IF NOT __ISVALIDREF(_stState)
THEN
  _eCheck                           := PROCESS_CHECK_STATE_REFERENCE_INVALID;
  RETURN;
END_IF
//-------------------------------------------------------------------------------------------------
//-------------------------------------------------------------------------------------------------
// plausibility checks
//-------------------------------------------------------------------------------------------------
IF NOT Check()
THEN
  RETURN;
END_IF
//-------------------------------------------------------------------------------------------------
//-------------------------------------------------------------------------------------------------
// Message device identification
//-------------------------------------------------------------------------------------------------
_stMsg.eDevice                      := e_Device.Process + TO_UINT(_nProcessId);
//-------------------------------------------------------------------------------------------------
//-------------------------------------------------------------------------------------------------
// XtsStation states:
//  - fb_ProcessCollector extends fb_StationCollector: 
//    --> cyclic call of States() for getting station masks
//
//  - sets bit for every XtsStation
//-------------------------------------------------------------------------------------------------
//
States();                           // collect XtsStation state information in masks
//-------------------------------------------------------------------------------------------------
//-------------------------------------------------------------------------------------------------
// process states
//-------------------------------------------------------------------------------------------------
CASE _stState.State
OF
  //-----------------------------------------------------------------------------------------------
  E_PROCESS_STATE.PROCESS_DISABLE:  // default wait state
    //-------------------------------------------------------------------------
    CASE _eStateProgress            // check if all my XtsStations are disabled
    OF
      E_PROGRESS.PROGRESS_INIT:
        IF (_wStateDisable = EXPT(2,_nStationCount)-1)                  // all stations in process range must be disabled at this point
        THEN
          _eStateProgress           := E_PROGRESS.PROGRESS_BUSY;

          IF (_MessageLevel = E_MessageType.eMessageVerbose)
          THEN
            _stMsg.eType            := E_MessageType.eMessageVerbose;
            _stMsg.eSubdevice       := e_Subdevice.Process_ProcessCollector_Cycle;
            _stMsg.iErrorNumber     := _nProcessId;
            _stMsg.sText            := concat(TO_STRING(_stState.State), ': ');
            _stMsg.sText            := concat(_stMsg.sText, TO_STRING(_eStateProgress));
            f_MessageSet(_stMsg);
          END_IF
        END_IF
    END_CASE
    //-------------------------------------------------------------------------
    CASE _eStateProgress            // check for process enable signal
    OF
      E_PROGRESS.PROGRESS_BUSY:
      CASE _stControl.Cmd                                               // check process command
      OF
        E_PROCESS_CTRL.PROCESS_ENABLE:
          _eCmd                     := _stControl.Cmd;                  // copy command from interface to local switch
          _wActivateStation         := _stControl.ActivateStation;      // on enabling of process, copy my active stations from interface

          _eStateProgress           := E_PROGRESS.PROGRESS_INIT;        // switch back sub state
          _stState.State            := E_PROCESS_STATE.PROCESS_ENABLE;  // switch to enable

          IF (_MessageLevel = E_MessageType.eMessageVerbose)
          THEN
            _stMsg.eType            := E_MessageType.eMessageVerbose;
            _stMsg.eSubdevice       := e_Subdevice.Process_ProcessCollector_Cycle;
            _stMsg.iErrorNumber     := _nProcessId;
            _stMsg.sText            := concat(TO_STRING(_stState.State), ': ');
            _stMsg.sText            := concat(_stMsg.sText, TO_STRING(_eStateProgress));
            f_MessageSet(_stMsg);
          END_IF
      END_CASE
    END_CASE
END_CASE
//-------------------------------------------------------------------------------------------------
//-------------------------------------------------------------------------------------------------
CASE _stState.State
OF
  //-----------------------------------------------------------------------------------------------
  E_PROCESS_STATE.PROCESS_ENABLE:   // wait here for process command "allow infeed"
    //-------------------------------------------------------------------------
    CASE _eStateProgress
    OF
      E_PROGRESS.PROGRESS_INIT:
        IF (_wStateEnable = _wActivateStation)                          // all active stations must be enabled
        THEN
          _eStateProgress           := E_PROGRESS.PROGRESS_BUSY;

          IF (_MessageLevel = E_MessageType.eMessageVerbose)
          THEN
            _stMsg.eType            := E_MessageType.eMessageVerbose;
            _stMsg.eSubdevice       := e_Subdevice.Process_ProcessCollector_Cycle;
            _stMsg.iErrorNumber     := _nProcessId;
            _stMsg.sText            := concat(TO_STRING(_stState.State), ': ');
            _stMsg.sText            := concat(_stMsg.sText, TO_STRING(_eStateProgress));
            f_MessageSet(_stMsg);
          END_IF
        END_IF
    END_CASE
    //-------------------------------------------------------------------------
    CASE _eStateProgress
    OF
      E_PROGRESS.PROGRESS_BUSY:
      // check command for further instructions
      CASE _stControl.Cmd
      OF
        E_PROCESS_CTRL.PROCESS_DISABLE:                                 // command decided to switch OFF  
          _eCmd                     := _stControl.Cmd;                  // copy command from interface
          _eStateProgress           := E_PROGRESS.PROGRESS_INIT;        // switch back sub state
          _stState.State            := E_PROCESS_STATE.PROCESS_DISABLE;

          IF (_MessageLevel = E_MessageType.eMessageVerbose)
          THEN
            _stMsg.eType            := E_MessageType.eMessageVerbose;
            _stMsg.eSubdevice       := e_Subdevice.Process_ProcessCollector_Cycle;
            _stMsg.iErrorNumber     := _nProcessId;
            _stMsg.sText            := concat(TO_STRING(_stState.State), ': ');
            _stMsg.sText            := concat(_stMsg.sText, TO_STRING(_eStateProgress));
            f_MessageSet(_stMsg);
          END_IF


        E_PROCESS_CTRL.PROCESS_STATIONS_INFEED:                          // command decided to allow checking the infeed into process
          _eStateProgress           := E_PROGRESS.PROGRESS_INIT;         // switch back sub state
          _stState.State            := E_PROCESS_STATE.PROCESS_STATIONS_INFEED;

          IF (_MessageLevel = E_MessageType.eMessageVerbose)
          THEN
            _stMsg.eType            := E_MessageType.eMessageVerbose;
            _stMsg.eSubdevice       := e_Subdevice.Process_ProcessCollector_Cycle;
            _stMsg.iErrorNumber     := _nProcessId;
            _stMsg.sText            := concat(TO_STRING(_stState.State), ': ');
            _stMsg.sText            := concat(_stMsg.sText, TO_STRING(_eStateProgress));
            f_MessageSet(_stMsg);
          END_IF
      END_CASE
    END_CASE
END_CASE
//-------------------------------------------------------------------------------------------------
//-------------------------------------------------------------------------------------------------
CASE _stState.State
OF
  //-----------------------------------------------------------------------------------------------
  E_PROCESS_STATE.PROCESS_STATIONS_INFEED:  // wait state for checking infeed command
    //-------------------------------------------------------------------------
    CASE _eStateProgress
    OF
      E_PROGRESS.PROGRESS_INIT:
        IF (_wStateEnter = _wActivateStation)                           // all active XtsStations must have mover waiting
        THEN
          // mover IDs are known by now --> Check _nMoverIdQueue for your plausibility checks
          _eStateProgress           := E_PROGRESS.PROGRESS_BUSY;

          IF (_MessageLevel = E_MessageType.eMessageVerbose)
          THEN
            _stMsg.eType            := E_MessageType.eMessageVerbose;
            _stMsg.eSubdevice       := e_Subdevice.Process_ProcessCollector_Cycle;
            _stMsg.iErrorNumber     := _nProcessId;
            _stMsg.sText            := concat(TO_STRING(_stState.State), ': ');
            _stMsg.sText            := concat(_stMsg.sText, TO_STRING(_eStateProgress));
            f_MessageSet(_stMsg);
          END_IF
        END_IF
    END_CASE
    //-------------------------------------------------------------------------
    CASE _eStateProgress
    OF
      E_PROGRESS.PROGRESS_BUSY:
      CASE _stControl.Cmd                                               // check command from interface
      OF
        E_PROCESS_CTRL.PROCESS_STATIONS_ENTER:
          _eCmd                     := _stControl.Cmd;                  // copy command to start infeed of movers

          _eStateProgress           := E_PROGRESS.PROGRESS_INIT;        // switch back sub state
          _stState.State            := E_PROCESS_STATE.PROCESS_START;

          IF (_MessageLevel = E_MessageType.eMessageVerbose)
          THEN
            _stMsg.eType            := E_MessageType.eMessageVerbose;
            _stMsg.eSubdevice       := e_Subdevice.Process_ProcessCollector_Cycle;
            _stMsg.iErrorNumber     := _nProcessId;
            _stMsg.sText            := concat(TO_STRING(_stState.State), ': ');
            _stMsg.sText            := concat(_stMsg.sText, TO_STRING(_eStateProgress));
            f_MessageSet(_stMsg);
          END_IF


        E_PROCESS_CTRL.PROCESS_STATIONS_SEND:
          _eCmd                     := _stControl.Cmd;                  // start skipping of process

          _eStateProgress           := E_PROGRESS.PROGRESS_INIT;        // switch back sub state
          _stState.State            := E_PROCESS_STATE.PROCESS_STATIONS_OUTFEED;

          IF (_MessageLevel = E_MessageType.eMessageVerbose)
          THEN
            _stMsg.eType            := E_MessageType.eMessageVerbose;
            _stMsg.eSubdevice       := e_Subdevice.Process_ProcessCollector_Cycle;
            _stMsg.iErrorNumber     := _nProcessId;
            _stMsg.sText            := concat(TO_STRING(_stState.State), ': ');
            _stMsg.sText            := concat(_stMsg.sText, TO_STRING(_eStateProgress));
            f_MessageSet(_stMsg);
          END_IF
      END_CASE
    END_CASE
END_CASE
//-------------------------------------------------------------------------------------------------
//-------------------------------------------------------------------------------------------------
CASE _stState.State
OF
  //-----------------------------------------------------------------------------------------------
  E_PROCESS_STATE.PROCESS_STATIONS_NEST:  // wait state before movers are positioned to next nest
    //-------------------------------------------------------------------------
    CASE _eStateProgress
    OF
      E_PROGRESS.PROGRESS_INIT:
        IF (_wStateNest = _wActivateStation)
        THEN
          _eStateProgress           := E_PROGRESS.PROGRESS_BUSY;

          IF (_MessageLevel = E_MessageType.eMessageVerbose)
          THEN
            _stMsg.eType            := E_MessageType.eMessageVerbose;
            _stMsg.eSubdevice       := e_Subdevice.Process_ProcessCollector_Cycle;
            _stMsg.iErrorNumber     := _nProcessId;
            _stMsg.sText            := concat(TO_STRING(_stState.State), ': ');
            _stMsg.sText            := concat(_stMsg.sText, TO_STRING(_eStateProgress));
            f_MessageSet(_stMsg);
          END_IF
        END_IF
    END_CASE
    //-------------------------------------------------------------------------
    CASE _eStateProgress
    OF
      E_PROGRESS.PROGRESS_BUSY:
      CASE _stControl.Cmd
      OF
        E_PROCESS_CTRL.PROCESS_STATIONS_ENTER:
          _eCmd                     := _stControl.Cmd;                  // copy command to start movement to next nest

          _eStateProgress           := E_PROGRESS.PROGRESS_INIT;        // switch back sub state
          _stState.State            := E_PROCESS_STATE.PROCESS_START;

          IF (_MessageLevel = E_MessageType.eMessageVerbose)
          THEN
            _stMsg.eType            := E_MessageType.eMessageVerbose;
            _stMsg.eSubdevice       := e_Subdevice.Process_ProcessCollector_Cycle;
            _stMsg.iErrorNumber     := _nProcessId;
            _stMsg.sText            := concat(TO_STRING(_stState.State), ': ');
            _stMsg.sText            := concat(_stMsg.sText, TO_STRING(_eStateProgress));
            f_MessageSet(_stMsg);
          END_IF
      END_CASE
    END_CASE
END_CASE
//-------------------------------------------------------------------------------------------------
//-------------------------------------------------------------------------------------------------
CASE _stState.State
OF
  //-----------------------------------------------------------------------------------------------
  E_PROCESS_STATE.PROCESS_START:    // wait state for movers to arrive
    //-------------------------------------------------------------------------
    CASE _eStateProgress
    OF
      E_PROGRESS.PROGRESS_INIT:
        IF (_wStateStart = _wActivateStation)                           // all active XtsStations have mover in standstill after infeed, process handshake may now start
        THEN
          // movers have arrived and are in standstill
          _eStateProgress           := E_PROGRESS.PROGRESS_BUSY;

          IF (_MessageLevel = E_MessageType.eMessageVerbose)
          THEN
            _stMsg.eType            := E_MessageType.eMessageVerbose;
            _stMsg.eSubdevice       := e_Subdevice.Process_ProcessCollector_Cycle;
            _stMsg.iErrorNumber     := _nProcessId;
            _stMsg.sText            := concat(TO_STRING(_stState.State), ': ');
            _stMsg.sText            := concat(_stMsg.sText, TO_STRING(_eStateProgress));
            f_MessageSet(_stMsg);
          END_IF
        END_IF
    END_CASE
    //-------------------------------------------------------------------------
    CASE _eStateProgress
    OF
      E_PROGRESS.PROGRESS_BUSY:
      CASE _stControl.Cmd
      OF
        E_PROCESS_CTRL.PROCESS_START:
          _eCmd                     := _stControl.Cmd;                  // first handshake for starting process

          _eStateProgress           := E_PROGRESS.PROGRESS_INIT;        // switch back sub state
          _stState.State            := E_PROCESS_STATE.PROCESS_DONE;

          IF (_MessageLevel = E_MessageType.eMessageVerbose)
          THEN
            _stMsg.eType            := E_MessageType.eMessageVerbose;
            _stMsg.eSubdevice       := e_Subdevice.Process_ProcessCollector_Cycle;
            _stMsg.iErrorNumber     := _nProcessId;
            _stMsg.sText            := concat(TO_STRING(_stState.State), ': ');
            _stMsg.sText            := concat(_stMsg.sText, TO_STRING(_eStateProgress));
            f_MessageSet(_stMsg);
          END_IF
      END_CASE
    END_CASE
END_CASE
//-------------------------------------------------------------------------------------------------
//-------------------------------------------------------------------------------------------------
CASE _stState.State
OF
  E_PROCESS_STATE.PROCESS_DONE:     // wait state for process done
    //-------------------------------------------------------------------------
    CASE _eStateProgress
    OF
      E_PROGRESS.PROGRESS_INIT:
        IF (_wStateDone = _wActivateStation)
        THEN
          // first handshake done
          _eStateProgress           := E_PROGRESS.PROGRESS_BUSY;

          IF (_MessageLevel = E_MessageType.eMessageVerbose)
          THEN
            _stMsg.eType            := E_MessageType.eMessageVerbose;
            _stMsg.eSubdevice       := e_Subdevice.Process_ProcessCollector_Cycle;
            _stMsg.iErrorNumber     := _nProcessId;
            _stMsg.sText            := concat(TO_STRING(_stState.State), ': ');
            _stMsg.sText            := concat(_stMsg.sText, TO_STRING(_eStateProgress));
            f_MessageSet(_stMsg);
          END_IF
        END_IF
    END_CASE
    //-------------------------------------------------------------------------
    CASE _eStateProgress
    OF
      E_PROGRESS.PROGRESS_BUSY:
      CASE _stControl.Cmd
      OF
        E_PROCESS_CTRL.PROCESS_DONE:
          _eCmd                     := _stControl.Cmd;                  // second handshake for finishing process

          _eStateProgress           := E_PROGRESS.PROGRESS_CHECK;       // check mover after process done
      END_CASE
    //-------------------------------------------------------------------------
      E_PROGRESS.PROGRESS_CHECK:
        IF (_wStateNest > 0)        // mover has to be worked again
        THEN
          _eStateProgress           := E_PROGRESS.PROGRESS_INIT;        // switch back sub state
          _stState.State            := E_PROCESS_STATE.PROCESS_STATIONS_NEST;

          IF (_MessageLevel = E_MessageType.eMessageVerbose)
          THEN
            _stMsg.eType            := E_MessageType.eMessageVerbose;
            _stMsg.eSubdevice       := e_Subdevice.Process_ProcessCollector_Cycle;
            _stMsg.iErrorNumber     := _nProcessId;
            _stMsg.sText            := concat(TO_STRING(_stState.State), ': ');
            _stMsg.sText            := concat(_stMsg.sText, TO_STRING(_eStateProgress));
            f_MessageSet(_stMsg);
          END_IF

        ELSIF (_wStateOut > 0)      // mover has to leave
        THEN
          _eStateProgress           := E_PROGRESS.PROGRESS_INIT;        // switch back sub state
          _stState.State            := E_PROCESS_STATE.PROCESS_STATIONS_OUTFEED;

          IF (_MessageLevel = E_MessageType.eMessageVerbose)
          THEN
            _stMsg.eType            := E_MessageType.eMessageVerbose;
            _stMsg.eSubdevice       := e_Subdevice.Process_ProcessCollector_Cycle;
            _stMsg.iErrorNumber     := _nProcessId;
            _stMsg.sText            := concat(TO_STRING(_stState.State), ': ');
            _stMsg.sText            := concat(_stMsg.sText, TO_STRING(_eStateProgress));
            f_MessageSet(_stMsg);
          END_IF
        END_IF
    END_CASE
END_CASE
//-------------------------------------------------------------------------------------------------
//-------------------------------------------------------------------------------------------------
CASE _stState.State
OF
  E_PROCESS_STATE.PROCESS_STATIONS_OUTFEED:   // wait state before movers are sent out
    //-------------------------------------------------------------------------
    CASE _eStateProgress
    OF
      E_PROGRESS.PROGRESS_INIT:
        IF (_wStateOut = _wActivateStation)
        THEN
          // all active stations want to send out mover
          // now is the time for you to have decided the TargetStation(s) and TargetMask(s)
          _eStateProgress           := E_PROGRESS.PROGRESS_BUSY;

          IF (_MessageLevel = E_MessageType.eMessageVerbose)
          THEN
            _stMsg.eType            := E_MessageType.eMessageVerbose;
            _stMsg.eSubdevice       := e_Subdevice.Process_ProcessCollector_Cycle;
            _stMsg.iErrorNumber     := _nProcessId;
            _stMsg.sText            := concat(TO_STRING(_stState.State), ': ');
            _stMsg.sText            := concat(_stMsg.sText, TO_STRING(_eStateProgress));
            f_MessageSet(_stMsg);
          END_IF
        END_IF
    END_CASE
    //-------------------------------------------------------------------------
    CASE _eStateProgress
    OF
      E_PROGRESS.PROGRESS_BUSY:     // now is the time to get/write target data
      CASE _stControl.Cmd
      OF
        E_PROCESS_CTRL.PROCESS_STATIONS_OUTFEED:  // before you start the outfeed of station, get/write target data on the outside. Use properties: TargetIndex; TargetMask
          _eCmd                     := _stControl.Cmd;
          _eStateProgress           := E_PROGRESS.PROGRESS_CHECK;       // check movers gone

          IF (_MessageLevel = E_MessageType.eMessageVerbose)
          THEN
            _stMsg.eType            := E_MessageType.eMessageVerbose;
            _stMsg.eSubdevice       := e_Subdevice.Process_ProcessCollector_Cycle;
            _stMsg.iErrorNumber     := _nProcessId;
            _stMsg.sText            := concat(TO_STRING(_stState.State), ': ');
            _stMsg.sText            := concat(_stMsg.sText, TO_STRING(_eStateProgress));
            f_MessageSet(_stMsg);
          END_IF
      END_CASE
    END_CASE
    //-------------------------------------------------------------------------
    CASE _eStateProgress
    OF
      E_PROGRESS.PROGRESS_CHECK:
        IF (_wStateOut = 0)         // all stations are empty, go back to start new infeed of movers
        THEN
          _eStateProgress           := E_PROGRESS.PROGRESS_INIT;        // switch back sub state
          _stState.State            := E_PROCESS_STATE.PROCESS_DISABLE; // switch back to disabled state

          IF (_MessageLevel = E_MessageType.eMessageVerbose)
          THEN
            _stMsg.eType            := E_MessageType.eMessageVerbose;
            _stMsg.eSubdevice       := e_Subdevice.Process_ProcessCollector_Cycle;
            _stMsg.iErrorNumber     := _nProcessId;
            _stMsg.sText            := concat(TO_STRING(_stState.State), ': ');
            _stMsg.sText            := concat(_stMsg.sText, TO_STRING(_eStateProgress));
            f_MessageSet(_stMsg);
          END_IF
        END_IF
    END_CASE
END_CASE
//-------------------------------------------------------------------------------------------------
// _eStateProgress information to process result
//-------------------------------------------------------------------------------------------------
_stState.Result                     := _eStateProgress;
//-------------------------------------------------------------------------------------------------
//-------------------------------------------------------------------------------------------------
// _eCheck information for plausibility checks
//-------------------------------------------------------------------------------------------------
_stState.Check                      := _eCheck;
//-------------------------------------------------------------------------------------------------
//-------------------------------------------------------------------------------------------------
// _eCmd - command switch
//-------------------------------------------------------------------------------------------------
Controls(_eCmd);                    // cyclic call for setting commands on XtsStations in process range
//-------------------------------------------------------------------------------------------------
//-------------------------------------------------------------------------------------------------
END_METHOD

METHOD PUBLIC Init : E_PROGRESS // clears all XtsSubstations, then disables all
VAR_INPUT
  Execute     : BOOL;
END_VAR
VAR_INST
  _nIndexStation        : UINT;
  _nErrorId             : UDINT;
  _eState               : E_PROGRESS;
END_VAR
//-----------------------------------------------------------------------------
IF NOT Execute 
THEN 
	_eState                       := E_PROGRESS.PROGRESS_INIT; 
END_IF 
//-----------------------------------------------------------------------------
IF NOT Check() 
THEN 
	Init                          := E_PROGRESS.PROGRESS_ERROR; 
	RETURN; 
END_IF
//-----------------------------------------------------------------------------
//-----------------------------------------------------------------------------
CASE _eState
OF
  E_PROGRESS.PROGRESS_INIT:
    IF Execute
    THEN
      _nIndexStation            := _nStationLast;
      _nErrorId                 := 0;
      _eState                   := E_PROGRESS.PROGRESS_BUSY;
      memset(ADR(_wTargetMask), 1, SIZEOF(_wTargetMask));

      _eCmd                     := E_PROCESS_CTRL.PROCESS_INIT;
      _stState.State            := E_PROCESS_STATE.PROCESS_INVALID;
      _eStateProgress           := E_PROGRESS.PROGRESS_INVALID;


      _stMsg.eType              := _MessageLevel;

      IF (_MessageLevel = E_MessageType.eMessageVerbose)
      THEN
        _stMsg.eSubdevice       := e_Subdevice.Process_ProcessCollector_Init;
        _stMsg.iErrorNumber     := _nIndexStation;
        _stMsg.sText            := concat('.Init: ', TO_STRING(_eState));
        f_MessageSet(_stMsg);
      END_IF
    END_IF
END_CASE
//-----------------------------------------------------------------------------
//-----------------------------------------------------------------------------
CASE _eState
OF
  E_PROGRESS.PROGRESS_BUSY:
    _StationCtrl[_nIndexStation].eCmd     := E_STATION_CTRL.STATION_INIT;
    _eState                     := E_PROGRESS.PROGRESS_PREPARE;

    IF (_MessageLevel = E_MessageType.eMessageVerbose)
    THEN
      _stMsg.eSubdevice         := e_Subdevice.Process_ProcessCollector_Init;
      _stMsg.iErrorNumber       := _nIndexStation;
      _stMsg.sText              := concat(TO_STRING(_StationCtrl[_nIndexStation].eCmd), ': ');
      _stMsg.sText              := concat(_stMsg.sText, TO_STRING(_eState));
      f_MessageSet(_stMsg);
    END_IF

  E_PROGRESS.PROGRESS_PREPARE:
    IF (_nIndexStation < _nStationFirst+1)
    THEN
      _eCmdOld                  :=
      _eCmd                     := E_PROCESS_CTRL.PROCESS_DISABLE;
      _nIndexStation            := _nStationFirst;
      _eState                   := E_PROGRESS.PROGRESS_STARTUP;
    ELSE
      IF (_StationState[_nIndexStation].eState = E_STATION_STATE.STATION_INIT)
      THEN
        _nIndexStation          := _nIndexStation - 1;
        _eState                 := E_PROGRESS.PROGRESS_BUSY;
      ELSE
        _eState                 := E_PROGRESS.PROGRESS_BUSY;
      END_IF
    END_IF

  E_PROGRESS.PROGRESS_STARTUP:
    _StationCtrl[_nIndexStation].eCmd     := E_STATION_CTRL.STATION_DISABLE;
    _eState                     := E_PROGRESS.PROGRESS_CHECK;

    IF (_MessageLevel = E_MessageType.eMessageVerbose)
    THEN
      _stMsg.eSubdevice         := e_Subdevice.Process_ProcessCollector_Init;
      _stMsg.iErrorNumber       := _nIndexStation;
      _stMsg.sText              := concat(TO_STRING(_StationCtrl[_nIndexStation].eCmd), ': ');
      _stMsg.sText              := concat(_stMsg.sText, TO_STRING(_eState));
      f_MessageSet(_stMsg);
    END_IF

  E_PROGRESS.PROGRESS_CHECK:
    IF NOT (_nIndexStation > _nStationLast-1)
    THEN
      IF (_StationState[_nIndexStation].eState = E_STATION_STATE.STATION_DISABLE)
      THEN
        _nIndexStation          := _nIndexStation + 1;
        _eState                 := E_PROGRESS.PROGRESS_STARTUP;
      END_IF
    ELSE
      // give back result
      _eState                   := E_PROGRESS.PROGRESS_DONE;

      // where were I?
      IF (_MessageLevel = E_MessageType.eMessageVerbose)
      THEN
        _stMsg.eSubdevice       := e_Subdevice.Process_ProcessCollector_Init;
        _stMsg.iErrorNumber     := _nProcessId;
        _stMsg.sText            := concat('.Clear: ', TO_STRING(_stState.State));
        f_MessageSet(_stMsg);
      END_IF

      // clear Cycle() state machine
      _stState.State            := E_PROCESS_STATE.PROCESS_DISABLE;
      _eStateProgress           := E_PROGRESS.PROGRESS_INIT;

      IF (_MessageLevel = E_MessageType.eMessageVerbose)
      THEN
        // init done
        _stMsg.eSubdevice       := e_Subdevice.Process_ProcessCollector_Init;
        _stMsg.iErrorNumber     := _nProcessId;
        _stMsg.sText            := concat('.Init: ', TO_STRING(_eState));
        f_MessageSet(_stMsg);
      END_IF
    END_IF
END_CASE
//-----------------------------------------------------------------------------
//-----------------------------------------------------------------------------

Init := _eState;
END_METHOD

PROPERTY MessageLevel : e_MessageType
GET
MessageLevel := _MessageLevel;
END_GET
SET
VAR
  _ix : uint;
END_VAR
_MessageLevel := MessageLevel;

IF NOT (_eCheck = E_PROCESS_CHECK.PROCESS_CHECK_DONE)
THEN
  RETURN;
ELSE
  FOR _ix := _nStationFirst TO _nStationLast
  DO
    GVL_MSG.MessageLevelStations[_ix]   := _MessageLevel;
  END_FOR
END_IF
END_SET
END_PROPERTY

PROPERTY MoverCountTotal : udint
GET
MoverCountTotal := _nMoverCountTotal;
END_GET
END_PROPERTY

PROPERTY MoverPerMinute : udint
GET
MoverPerMinute := _AllStationMoverPerMinute;
END_GET
END_PROPERTY

PROPERTY ProcessCtrl : reference to st_process_ctrl
GET
ProcessCtrl REF= _stControl;
END_GET
SET
_stControl ref= ProcessCtrl;
END_SET
END_PROPERTY

PROPERTY ProcessId : E_INSTANCE
GET
Processid := _nProcessId;
END_GET
SET
_nProcessId := ProcessId;
END_SET
END_PROPERTY

PROPERTY ProcessState : reference to st_process_state
GET
ProcessState REF= _stState;
END_GET
SET
_stState ref= ProcessState;
END_SET
END_PROPERTY

PROPERTY TargetIndex : ARRAY[1..SIZEOF(T_PROCESS)*8] OF USINT
GET
TargetIndex := _nTargetIndex;
END_GET
SET
_nTargetIndex := TargetIndex;
END_SET
END_PROPERTY

PROPERTY TargetMask : ARRAY[1..SIZEOF(T_PROCESS)*8] OF BYTE
GET
TargetMask := _wTargetMask;
END_GET
SET
_wTargetMask := TargetMask;
END_SET
END_PROPERTY

METHOD Template : E_PROGRESS
VAR_INPUT
  Execute     : BOOL;
END_VAR
VAR_INST
  _nErrorId   : UDINT;
  _eState     : E_PROGRESS;
END_VAR
//-----------------------------------------------------------------------------
IF NOT Execute 
THEN 
	_eState                       := E_PROGRESS.PROGRESS_INIT; 
END_IF 
//-----------------------------------------------------------------------------
IF NOT Check() 
THEN 
	Template_1                    := E_PROGRESS.PROGRESS_ERROR; 
	RETURN; 
END_IF
//-----------------------------------------------------------------------------
//-----------------------------------------------------------------------------
CASE _eState
OF
  E_PROGRESS.PROGRESS_INIT:
    IF Execute
    THEN
      _nErrorId                 := 0;

      _eState                   := E_PROGRESS.PROGRESS_BUSY;
    END_IF
END_CASE
//-----------------------------------------------------------------------------
//-----------------------------------------------------------------------------
CASE _eState
OF
  E_PROGRESS.PROGRESS_BUSY:
    _eState                     := E_PROGRESS.PROGRESS_PREPARE;
END_CASE
//-----------------------------------------------------------------------------
//-----------------------------------------------------------------------------
CASE _eState
OF
  E_PROGRESS.PROGRESS_PREPARE:

    IF (.Error)
    THEN
      _eState                   := E_PROGRESS.PROGRESS_ERROR;
      _nErrorId                 := 


    ELSIF (.Done)
    THEN
      _eState                   := E_PROGRESS.;

    END_IF
END_CASE
//-----------------------------------------------------------------------------
//-----------------------------------------------------------------------------

Template_1                      := _eState;
END_METHOD

END_FUNCTION_BLOCK

// ---- XTS/XtsStation/fb_Station.TcPOU
//---------------------------------------------------------------------------------------------------------------
//
//  HAUD 2023.03.07
//
//  - XTS_TRANSPORT_LAYER
//
//  fb_Station
//  - handshake with extern control for mover transport through station
//
//---------------------------------------------------------------------------------------------------------------
// This SOFTWARE is provided as an Exemple by THE PROVIDER "as is" and "with all faults." THE PROVIDER makes no 
// representations or warranties of any kind concerning the safety, suitability, lack of viruses, inaccuracies, 
// typographical errors, or other harmful components of this SOFTWARE. There are inherent dangers in the use of 
// any software, and you are solely responsible for determining whether this SOFTWARE is compatible with your 
// equipment and other software installed on your equipment. You are also solely responsible for the protection 
// of your equipment and backup of your data, and THE PROVIDER will not be liable for any damages you may suffer 
// in connection with using, modifying, or distributing this SOFTWARE.
//---------------------------------------------------------------------------------------------------------------
FUNCTION_BLOCK fb_Station IMPLEMENTS I_XtsTransport_Station
VAR
  _nStationId                 : UINT;         // why is Gamora?

  _sState                     : STRING(255);  // additional output for Check()

  _eInitList                  : E_PROGRESS;   // linked list initialization progress

  _eFatalError                : E_STATION_STATE;

  // pointer to all stations
  _stCtrl                     : REFERENCE TO ARRAY[1..MAX_STATION]  OF ST_STATION_CTRL;
  _stState                    : REFERENCE TO ARRAY[1..MAX_STATION]  OF ST_STATION_STATE;

  // local copy of command
  _eCmd,
  _eCmdOld                    : E_STATION_CTRL;

  _ItfStation                 : REFERENCE TO ARRAY[1..MAX_STATION]  OF I_Station_LinkedList;  // access to all stations lists
  _ItfMover                   : REFERENCE TO ARRAY[1..MAX_MOVER]    OF I_XtsTransport_Mover;  // access to mover methods

  // station related data
  _rMoverOffset               : REFERENCE TO ARRAY[1..MAX_STATION]  OF T_NEST_OFFSET;         // static offsets for station
  _stParameter                : REFERENCE TO ARRAY[1..MAX_STATION]  OF ST_STATION_PARAMETER;  // station parameter (where, how fast, how many stops)

  // mover axis ref for info
  _Mover                      : REFERENCE TO ARRAY[1..MAX_MOVER]    OF AXIS_REF;              // read from AXIS_REF

  // linked list result struct
  _stListEnter,
  _stListTarget,
  _stListDelete               : ST_STATION_LIST_RESULT;   // struct with result and ticket data

  _stMoverDataSend,
  _stMoverData                : ST_STATION_MOVER_DATA;    // mover ticket data

  _stInfeed,
  _stOutfeed                  : ST_MOVE_DATA;             // position and dynamic constraints of movement

  // work vars
  _Result                     : E_PROGRESS;
  _eStateProgress             : E_PROGRESS;

  _nNest,
  _nMoverDetected,
  _ix                         : UINT;

  _rModActPosFetch            : LREAL;
  _stMsg                      : ST_Message;
  _eMessageLevel              : E_MessageType;
  _bMatchMessageLevel         : BOOL := TRUE;   // TRUE --> Mover in Station commands have equal message level as station
END_VAR

METHOD PRIVATE Check : BOOL
VAR_INPUT
END_VAR
IF NOT (_nStationId > 0) OR
       (_nStationId > MAX_STATION)
THEN
  _sState                     := 'invalid nStationId';
  RETURN;
END_IF

IF NOT __ISVALIDREF(_stCtrl)
THEN
  _sState                     := '_stCtrl: missing pointer';
  RETURN;
END_IF

IF NOT __ISVALIDREF(_stState)
THEN
  _sState                     := '_stState: missing pointer';
  RETURN;
END_IF

IF NOT __ISVALIDREF(_ItfStation)
THEN
  _sState                     := '_ItfStation: missing interface';
  RETURN;
END_IF

IF NOT __ISVALIDREF(_ItfMover)
THEN
  _sState                     := '_ItfMover: missing interface';
  RETURN;
END_IF

IF NOT __ISVALIDREF(_rMoverOffset)
THEN
  _sState                     := '_rMoverOffset: missing pointer';
  RETURN;
END_IF

IF NOT __ISVALIDREF(_stParameter)
THEN
  _sState                     := '_stParameter: missing pointer';
  RETURN;
END_IF

IF NOT __ISVALIDREF(_Mover)
THEN
  _sState                     := '_Mover: missing pointer';
  RETURN;
END_IF


_sState                       := 'CHECK_DONE';
Check                         := TRUE;
END_METHOD

PROPERTY Ctrl : reference to ARRAY[1..MAX_STATION] OF ST_STATION_CTRL
SET
_stCtrl ref= Ctrl;
END_SET
END_PROPERTY

METHOD Cycle
//-----------------------------------------------------------------------------
//-----------------------------------------------------------------------------
// check pointer and interface
//-----------------------------------------------------------------------------
IF NOT Check() THEN RETURN; END_IF
//-----------------------------------------------------------------------------
//-----------------------------------------------------------------------------
// set message device ID
//-----------------------------------------------------------------------------
_stMsg.eDevice                        := e_Device.XtsStation + _nStationId;
//-----------------------------------------------------------------------------
//-----------------------------------------------------------------------------
// log command change
//-----------------------------------------------------------------------------
_eCmd                                 := _stCtrl[_nStationId].eCmd;
IF (_eCmd <> _eCmdOld)
THEN
  _eCmdOld                            := _eCmd;

  _stMsg.eType                        := E_MessageType.eMessageInfo;
  _stMsg.eSubdevice                   := StationControl;
  _stMsg.iErrorNumber                 := 0;
  _stMsg.sText                        := TO_STRING(_eCmd);

  IF (_eMessageLevel > E_MessageType.eMessageWarning)
  THEN
    f_MessageSet(_stMsg);
  END_IF
END_IF
//-----------------------------------------------------------------------------
//-----------------------------------------------------------------------------
// clear station on demand
//-----------------------------------------------------------------------------
CASE _stCtrl[_nStationId].eCmd
OF
  E_STATION_CTRL.STATION_INIT:        // commanded init from cyclic interface
    _eInitList                        := Init();
    _stState[_nStationId].rMoverModPos:= 0.0;
    _stState[_nStationId].nQueue      := TO_USINT(_ItfStation[_nStationId].Count);
    RETURN;
END_CASE
//-----------------------------------------------------------------------------
//-----------------------------------------------------------------------------
// station startup and init states
//-----------------------------------------------------------------------------
CASE _stState[_nStationId].eState
OF
  E_STATION_STATE.STATION_NO_INIT:    // startup state in first PLC cycle, init linked list required
    _eInitList                        := Init();

  E_STATION_STATE.STATION_INIT:       // switch state as reserve for anything you might add here
    _stState[_nStationId].eState      := E_STATION_STATE.STATION_DISABLE;
END_CASE
//-----------------------------------------------------------------------------
//-----------------------------------------------------------------------------
//  station disabled after init 
//  wait for command to enable
//  return state after a mover has left station
//  fall back state before entry was allowed and you decided to disable
//-----------------------------------------------------------------------------
CASE _stState[_nStationId].eState
OF
  E_STATION_STATE.STATION_DISABLE:
    IF (_stCtrl[_nStationId].eCmd = E_STATION_CTRL.STATION_ENABLE)
    THEN
      _stState[_nStationId].eState    := E_STATION_STATE.STATION_ENABLE;
    END_IF


  E_STATION_STATE.STATION_ENABLE:     // enable state is detectable on the interface for one cycle only
                                      // double check commanded enable and clear work vars
    IF (_stCtrl[_nStationId].eCmd = E_STATION_CTRL.STATION_ENABLE)
    THEN
      memset(ADR(_stListEnter),    0, SIZEOF(_stListEnter));

      _eStateProgress                 := E_PROGRESS.PROGRESS_INIT;  // substate for procedures within one state
      _stState[_nStationId].eState    := E_STATION_STATE.STATION_DETECT_MOVER;  // switch to mover detection

      IF (_eMessageLevel = E_MessageType.eMessageVerbose)
      THEN
        _stMsg.eType                  := _eMessageLevel;
        LogState(_stMsg.eType);
      END_IF
    END_IF
END_CASE
//-----------------------------------------------------------------------------
//-----------------------------------------------------------------------------
//  detection state
//   - wait until mover data is entered into list
//
//  check for disable command; fall back to disabled state
//  check linked list for new entry; proceed to request infeed of mover
//-----------------------------------------------------------------------------
CASE _stState[_nStationId].eState
OF
  E_STATION_STATE.STATION_DETECT_MOVER:// wait state for mover detection
    CASE _eStateProgress
    OF
      E_PROGRESS.PROGRESS_INIT:
        IF (_stCtrl[_nStationId].eCmd = E_STATION_CTRL.STATION_DISABLE) // check for commanded disable
        THEN
          IF (_eMessageLevel = E_MessageType.eMessageVerbose)
          THEN
            _stMsg.eType              := E_MessageType.eMessageVerbose;
            _stMsg.eSubdevice         := Stationstate;
            _stMsg.iErrorNumber       := _stState[_nStationId].nMoverId;
            _stMsg.sText              := concat(TO_STRING(_stState[_nStationId].eState), ': ');
            _stMsg.sText              := concat(_stMsg.sText, TO_STRING(E_STATION_STATE.STATION_DISABLE));
            f_MessageSet(_stMsg);
          END_IF
          _stState[_nStationId].eState      := E_STATION_STATE.STATION_DISABLE; // go back and wait, no matter the queue

        ELSIF (_ItfStation[_nStationId].Count > 0)
        THEN
          // someone entered something in my list
          _stListEnter                := _ItfStation[_nStationId].GetHead();
          _eStateProgress             := E_PROGRESS.PROGRESS_BUSY;  // go check list result data

          IF (_eMessageLevel > E_MessageType.eMessageWarning)
          THEN
            _stMsg.eType              := E_MessageType.eMessageInfo;
            _stMsg.eSubdevice         := Stationstate;
            _stMsg.iErrorNumber       := _stState[_nStationId].nMoverId;
            _stMsg.sText              := concat(TO_STRING(_stState[_nStationId].eState), ': ');
            _stMsg.sText              := concat(_stMsg.sText, TO_STRING(_eStateProgress));
            f_MessageSet(_stMsg);
          END_IF
        END_IF
    END_CASE
    CASE _eStateProgress
    OF
      E_PROGRESS.PROGRESS_BUSY:
        IF (_stListEnter.wState = 0)  // GetHead() without error
        THEN
          _stMsg.eType                := E_MessageType.eMessageVerbose;
          _stMsg.eSubdevice           := e_Subdevice.StationGetHead;
          _stMsg.iErrorNumber         := _stListEnter.stData.nMoverId;
          _stMsg.sText                := '';
          IF (_eMessageLevel = E_MessageType.eMessageVerbose)
          THEN
            f_MessageSet(_stMsg);
          END_IF

          // list is giving head as result
          _stMoverData                := _stListEnter.stData; // copy ticket from list result
          _eStateProgress             := E_PROGRESS.PROGRESS_PREPARE; // go check plausibility of ticket

          IF (_eMessageLevel = E_MessageType.eMessageVerbose)
          THEN
            _stMsg.eType              := E_MessageType.eMessageVerbose;
            _stMsg.eSubdevice         := Stationstate;
            _stMsg.iErrorNumber       := _stState[_nStationId].nMoverId;
            _stMsg.sText              := concat(TO_STRING(_stState[_nStationId].eState), ': ');
            _stMsg.sText              := concat(_stMsg.sText, TO_STRING(_eStateProgress));
            f_MessageSet(_stMsg);
          END_IF
        ELSE
          // the thing that must not be: GetHead() with error
          _stState[_nStationId].eState      := E_STATION_STATE.STATION_ERROR_LIST_GET_HEAD_FAULT; // fatal error

          _stMsg.eType                      := E_MessageType.eMessageError;
          LogState(_stMsg.eType);
        END_IF
    END_CASE
    CASE _eStateProgress
    OF
      E_PROGRESS.PROGRESS_PREPARE:    // check ticket (list entry)
        // check target assignement
        IF NOT (_stMoverData.nTargetStation = _nStationId)
        THEN
          // for whom the mover calls
          // wrong address, right mover?
          _stState[_nStationId].eState      := E_STATION_STATE.STATION_ERROR_LIST_STATION_ID_WRONG; // ctrl has to fix this, go tell ctrl

          _stMsg.eType                      := E_MessageType.eMessageWarning;
          LogState(_stMsg.eType);
        ELSE
          // it's a me
          _nMoverDetected                   := _stMoverData.nMoverId;

          IF (_nMoverDetected < 1) OR
             (_nMoverDetected > MAX_MOVER)
          THEN
            // out of range the mover must not be
            _stState[_nStationId].eState    := E_STATION_STATE.STATION_ERROR_LIST_MOVER_ID_INVALID; // fatal error

            _stMsg.eType                    := E_MessageType.eMessageError;
            LogState(_stMsg.eType);
          ELSE
            memset(ADR(_stListDelete),   0, SIZEOF(_stListDelete)); // clear work var
            _eStateProgress                 := E_PROGRESS.PROGRESS_INIT; // clear progress for next station state

            // prepare station state for new mover
            _stState[_nStationId].nMoverId  := TO_USINT(_nMoverDetected); // who is waiting to enter
            _stState[_nStationId].nMask     := _stMoverData.nMask;        // how many stops have to be made
            _stState[_nStationId].eState    := E_STATION_STATE.STATION_MOVER_ENTER; // go ask for permission to enter

            IF (_eMessageLevel > E_MessageType.eMessageWarning)
            THEN
              _stMsg.eType            := E_MessageType.eMessageInfo;
              _stMsg.eSubdevice       := Stationstate;
              _stMsg.iErrorNumber     := _stState[_nStationId].nMoverId;
              _stMsg.sText            := concat(TO_STRING(_stState[_nStationId].eState), ': ');
              _stMsg.sText            := concat(_stMsg.sText, TO_STRING(_eStateProgress));
              f_MessageSet(_stMsg);
            END_IF
          END_IF
        END_IF
    END_CASE
END_CASE
//-----------------------------------------------------------------------------
//-----------------------------------------------------------------------------
// enter into station state
//  last check for disable command; fall back to disabled state
//  check for command to enter; prepare moverment, start movement
//  check for command to skip; prepare movement, switch to outfeed state
//-----------------------------------------------------------------------------
CASE _stState[_nStationId].eState
OF
  E_STATION_STATE.STATION_MOVER_ENTER:          // requesting permission for mover to enter station
    CASE _eStateProgress
    OF
      E_PROGRESS.PROGRESS_INIT:

        CASE _stCtrl[_nStationId].eCmd
        OF
          E_STATION_CTRL.STATION_DISABLE:       // control decided to disable, mover will wait
            _stState[_nStationId].eState    := E_STATION_STATE.STATION_DISABLE;

            IF (_eMessageLevel = E_MessageType.eMessageVerbose)
            THEN
              _stMsg.eType                  := _eMessageLevel;
              LogState(_stMsg.eType);
            END_IF

          E_STATION_CTRL.STATION_MOVER_ENTER:   // control decided to let mover enter
            _nNest                    := 1;     // default nest/PosStop[1]
            _eStateProgress           := E_PROGRESS.PROGRESS_BUSY;

            IF (_eMessageLevel = E_MessageType.eMessageVerbose)
            THEN
              _stMsg.eType            := E_MessageType.eMessageVerbose;
              _stMsg.eSubdevice       := Stationstate;
              _stMsg.iErrorNumber     := _stState[_nStationId].nMoverId;
              _stMsg.sText            := concat(TO_STRING(_stState[_nStationId].eState), ': ');
              _stMsg.sText            := concat(_stMsg.sText, TO_STRING(_eStateProgress));
              f_MessageSet(_stMsg);
            END_IF

            FOR _ix := 1 TO _stParameter[_nStationId].nConfiguredStopCount
            DO
              IF GetBitWord(_stMoverData.nMask, _ix-1)
              THEN
                _nNest                := _ix;
                EXIT;
              END_IF
            END_FOR

          E_STATION_CTRL.STATION_MOVER_SEND:    // control decided to send mover away
            _stOutfeed.rDistance          := _stParameter[_nStationId].rReleaseDistance;
            _stState[_nStationId].eState  := E_STATION_STATE.STATION_MOVER_OUT;

            IF (_eMessageLevel = E_MessageType.eMessageVerbose)
            THEN
              _stMsg.eType                := _eMessageLevel;
              LogState(_stMsg.eType);
            END_IF
        END_CASE
    END_CASE
    CASE _eStateProgress
    OF
      E_PROGRESS.PROGRESS_BUSY:
        MoveData();                   // prepare movement into station

        // check if infeed movement has to cross modulo turn
        _rModActPosFetch              := _Mover[_stMoverData.nMoverId].NcToPlc.ModuloActPos;

        IF (_rModActPosFetch > _stInfeed.rPos + _stParameter[_nStationId].rReleaseDistance)
        THEN
          _stInfeed.rPos              := _stInfeed.rPos + TO_REAL(_ItfMover[_stMoverData.nMoverId].RailLength);
        END_IF

        _stState[_nStationId].eState  := E_STATION_STATE.STATION_MOVER_IN_TARGET;

        IF (_eMessageLevel = E_MessageType.eMessageVerbose)
        THEN
          _stMsg.eType                := _eMessageLevel;
          LogState(_stMsg.eType);
        END_IF
    END_CASE
END_CASE
//-----------------------------------------------------------------------------
//-----------------------------------------------------------------------------
// move into station state
//  wait for movement to be done; mover in position and standstill
//    switch state to process handshake
//-----------------------------------------------------------------------------
CASE _stState[_nStationId].eState
OF
  E_STATION_STATE.STATION_MOVER_IN_TARGET:
    _ItfMover[_stMoverData.nMoverId].MessageLevel := SEL(_bMatchMessageLevel, E_MessageType.eMessageError, _eMessageLevel);

    _Result := _ItfMover[_stState[_nStationId].nMoverId].MoveToPosCa(TRUE, _stInfeed);

    IF (_Result = E_PROGRESS.PROGRESS_DONE)
    THEN
      // mother! has arrived
      _ItfMover[_stState[_nStationId].nMoverId].MoveToPosCa(FALSE, _stInfeed);
      _stState[_nStationId].eState    := E_STATION_STATE.STATION_PROCESS_START;

      IF (_eMessageLevel > E_MessageType.eMessageWarning)
      THEN
        _stMsg.eType                  := E_MessageType.eMessageInfo;
        LogState(_stMsg.eType);
      END_IF
    ELSE
      IF (_Result = E_PROGRESS.PROGRESS_ERROR)
      THEN
        _ItfMover[_stState[_nStationId].nMoverId].MoveToPosCa(FALSE, _stInfeed);
        _stState[_nStationId].eState  := E_STATION_STATE.STATION_ERROR_INFEED_ERROR; // ctrl has to fix this, go tell ctrl

        _stMsg.eType                  := E_MessageType.eMessageError;
        LogState(_stMsg.eType);
      END_IF 
    END_IF
END_CASE
//-----------------------------------------------------------------------------
//-----------------------------------------------------------------------------
// process handshake state
//  clear bit in mask
//-----------------------------------------------------------------------------
CASE _stState[_nStationId].eState
OF
  E_STATION_STATE.STATION_PROCESS_START:
    IF (_stCtrl[_nStationId].eCmd = E_STATION_CTRL.STATION_PROCESS_START) OR  // double handshake, your choice
       (_stCtrl[_nStationId].eCmd = E_STATION_CTRL.STATION_PROCESS_DONE)  OR  // single handshake, your choice
       (_stCtrl[_nStationId].eCmd = E_STATION_CTRL.STATION_MOVER_OUT)         // quick release, mask is not checked, mover will be sent out
    THEN
      // clear bit in mask when started/done
      _stState[_nStationId].nMask     := TO_USINT(DelBitWord(TO_WORD(_stState[_nStationId].nMask), _nNest-1));
      _stState[_nStationId].eState    := E_STATION_STATE.STATION_PROCESS_DONE;

      IF (_eMessageLevel = E_MessageType.eMessageVerbose)
      THEN
        _stMsg.eType                  := _eMessageLevel;
        LogState(_stMsg.eType);
      END_IF
    END_IF
END_CASE
//-----------------------------------------------------------------------------
//-----------------------------------------------------------------------------
CASE _stState[_nStationId].eState
OF
  E_STATION_STATE.STATION_PROCESS_DONE:
    IF (_stCtrl[_nStationId].eCmd = E_STATION_CTRL.STATION_PROCESS_DONE)
    THEN
      _stState[_nStationId].eState    := E_STATION_STATE.STATION_CHECK;

    ELSIF (_stCtrl[_nStationId].eCmd = E_STATION_CTRL.STATION_MOVER_OUT)
    THEN
      _stState[_nStationId].eState    := E_STATION_STATE.STATION_MOVER_OUT;
    END_IF
END_CASE
//-----------------------------------------------------------------------------
//-----------------------------------------------------------------------------
// check state if the mover has to move to another nest or must leave station
//-----------------------------------------------------------------------------
CASE _stState[_nStationId].eState
OF
  E_STATION_STATE.STATION_CHECK:
    IF (_stState[_nStationId].nMask = 0)
    THEN
      // mover has to leave
      _stState[_nStationId].eState    := E_STATION_STATE.STATION_MOVER_OUT;

      IF (_eMessageLevel = E_MessageType.eMessageVerbose)
      THEN
        _stMsg.eType                  := _eMessageLevel;
        LogState(_stMsg.eType);
      END_IF
    ELSE
      // _stState[_nStationId].nMask <> 0
      FOR _ix := 1 TO MAX_STATION_NEST
      DO
        IF NOT (_ix > _stParameter[_nStationId].nConfiguredStopCount)
        THEN
          IF GetBitWord(_stState[_nStationId].nMask, _ix-1)
          THEN
            // more work to do
            _stState[_nStationId].eState  := E_STATION_STATE.STATION_CHECK_NEST;
            _nNest                        := _ix; // index to move to

            IF (_eMessageLevel = E_MessageType.eMessageVerbose)
            THEN
              _stMsg.eType                := _eMessageLevel;
              LogState(_stMsg.eType);
            END_IF
            EXIT;
          END_IF
        ELSE
          IF GetBitWord(_stState[_nStationId].nMask, _ix-1)
          THEN
            // not configured, not worked
            _stMsg.eType              := E_MessageType.eMessageWarning;
            _stMsg.eSubdevice         := Stationstate;
            _stMsg.iErrorNumber       := _ix;
            _stMsg.sText              := concat(TO_STRING(_stState[_nStationId].eState), ': ');
            _stMsg.sText              := concat(_stMsg.sText, Tc2_Utilities.BYTE_TO_BINSTR(_stState[_nStationId].nMask, TO_INT(MAX_STATION_NEST)));
            IF (_eMessageLevel > E_MessageType.eMessageError)
            THEN
              f_MessageSet(_stMsg);
            END_IF

            _stState[_nStationId].nMask := TO_USINT(DelBitWord(TO_WORD(_stState[_nStationId].nMask), _ix-1));
          END_IF
        END_IF
      END_FOR
    END_IF
END_CASE
//-----------------------------------------------------------------------------
//-----------------------------------------------------------------------------
// wait state before movement to next nest has to be started
//-----------------------------------------------------------------------------
CASE _stState[_nStationId].eState
OF
  E_STATION_STATE.STATION_CHECK_NEST:
    IF (_stCtrl[_nStationId].eCmd = E_STATION_CTRL.STATION_MOVER_ENTER)
    THEN
      MoveData();
      _stState[_nStationId].eState    := E_STATION_STATE.STATION_MOVER_IN_TARGET;
  
      IF (_eMessageLevel = E_MessageType.eMessageVerbose)
      THEN
        _stMsg.eType                  := _eMessageLevel;
        LogState(_stMsg.eType);
      END_IF
    END_IF
END_CASE
//-----------------------------------------------------------------------------
//-----------------------------------------------------------------------------
// wait state for outfeed of mover
//  check ctrl data, target must be plausible, nTargetStation is what you have to set
//-----------------------------------------------------------------------------
CASE _stState[_nStationId].eState
OF
  E_STATION_STATE.STATION_MOVER_OUT:
    IF (_stCtrl[_nStationId].eCmd = E_STATION_CTRL.STATION_MOVER_OUT)
    THEN
      IF (_stCtrl[_nStationId].nTargetStation < 1) OR  
         (_stCtrl[_nStationId].nTargetStation > MAX_STATION)
      THEN
        _stState[_nStationId].eState  := E_STATION_STATE.STATION_ERROR_OUTFEED_TARGET_INVALID; // ctrl has to fix this, go tell ctrl

        _stMsg.eType                  := E_MessageType.eMessageError;
        LogState(_stMsg.eType);
      ELSE
        _stListDelete                 := _ItfStation[_nStationId].RemoveHeadValue(); // delete mover data in stations linked list


        IF (_stListDelete.wState <> 0)
        THEN
        // deleting mover in list was NOT successful
          _stState[_nStationId].eState:= E_STATION_STATE.STATION_ERROR_LIST_REMOVE_HEAD_FAULT; // fatal error

          _stMsg.eType                := E_MessageType.eMessageError;
          LogState(_stMsg.eType);

        ELSE
        // mover data successfully deleted
          _stMsg.eType                := E_MessageType.eMessageVerbose;
          _stMsg.eSubdevice           := e_Subdevice.StationRemoveHeadValue;
          _stMsg.iErrorNumber         := _stState[_nStationId].nMoverId;
          _stMsg.sText                := '';
          IF (_eMessageLevel = E_MessageType.eMessageVerbose)
          THEN
            f_MessageSet(_stMsg);
          END_IF

          memset(ADR(_stListTarget),   0, SIZEOF(_stListTarget)); // clear debug var

          // prepare movement and switch state to start movement
          MoverOut();
          _stState[_nStationId].eState  := E_STATION_STATE.STATION_MOVER_RELEASE;

          IF (_eMessageLevel > E_MessageType.eMessageWarning)
          THEN
            _stMsg.eType                := E_MessageType.eMessageInfo;
            LogState(_stMsg.eType);
          END_IF
        END_IF
      END_IF
    END_IF
END_CASE
//-----------------------------------------------------------------------------
//-----------------------------------------------------------------------------
// ckeck if mover has left the station
//  enter mover data into list of target station
//-----------------------------------------------------------------------------
CASE _stState[_nStationId].eState
OF
  E_STATION_STATE.STATION_MOVER_RELEASE:
    _ItfMover[_stMoverData.nMoverId].MessageLevel := SEL(_bMatchMessageLevel, E_MessageType.eMessageError, _eMessageLevel);

    _Result                           := _ItfMover[_stMoverDataSend.nMoverId].SendToModuloPosCa(TRUE, _stOutfeed);

    IF (_Result = E_PROGRESS.PROGRESS_DONE)
    THEN
      // regular outfeed
      _stState[_nStationId].eState    := E_STATION_STATE.STATION_MOVER_WRITE_TARGET;

    ELSIF (_stCtrl[_nStationId].eCmd = E_STATION_CTRL.STATION_MOVER_GONE) // in case outfeed has to be terminated by ctrl
    THEN
      // in order to finish the outfeed, ticket data has to be written to target station
      _stState[_nStationId].eState    := E_STATION_STATE.STATION_MOVER_WRITE_TARGET;

    ELSIF (_Result = E_PROGRESS.PROGRESS_ERROR)
    THEN
      _stState[_nStationId].eState    := E_STATION_STATE.STATION_ERROR_OUTFEED_ERROR; // ctrl has to fix this, go tell ctrl
      _stMsg.eType                    := E_MessageType.eMessageError;
      LogState(_stMsg.eType);
    END_IF
END_CASE
//-----------------------------------------------------------------------------
//-----------------------------------------------------------------------------
// write mover ticket in target station list
//
//-----------------------------------------------------------------------------
CASE _stState[_nStationId].eState
OF
  E_STATION_STATE.STATION_MOVER_WRITE_TARGET:
    // add entry in target station list
    _stListTarget                   := _ItfStation[_stMoverDataSend.nTargetStation].AddTailValue(_stMoverDataSend);
  
    IF (_stListTarget.wState <> 0)
    THEN
    // adding mover in target list was NOT successful
      _stState[_nStationId].eState  := E_STATION_STATE.STATION_ERROR_LIST_ADD_TAIL_FAULT; // fatal error
      _stMsg.eType                  := E_MessageType.eMessageError;
      LogState(_stMsg.eType);
  
    ELSE
    // mover data successfully added to target station list
      IF (_eMessageLevel > E_MessageType.eMessageWarning)
      THEN
        _stMsg.eType                := E_MessageType.eMessageInfo;
        _stMsg.eSubdevice           := e_Subdevice.StationAddTail;
        _stMsg.iErrorNumber         := _stState[_nStationId].nMoverId;
        _stMsg.sText                := concat('TargetStation: ', TO_STRING(_stListTarget.stData.nTargetStation));
        f_MessageSet(_stMsg);
      END_IF
      _ItfMover[_stMoverDataSend.nMoverId].SendToModuloPosCa(FALSE, _stOutfeed);
  
      _stState[_nStationId].eState  := E_STATION_STATE.STATION_MOVER_GONE; // go tell ctrl that station is empty
  
      IF (_eMessageLevel = E_MessageType.eMessageVerbose)
      THEN
        _stMsg.eType                := _eMessageLevel;
        LogState(_stMsg.eType);
      END_IF
    END_IF
END_CASE
//-----------------------------------------------------------------------------
//-----------------------------------------------------------------------------
// check handshake for empty station
//  switch back station state for new mover to be able to enter
//-----------------------------------------------------------------------------
CASE _stState[_nStationId].eState
OF
  E_STATION_STATE.STATION_MOVER_GONE:

    memset(ADR(_stMoverData),  0, SIZEOF(_stMoverData));

    _stState[_nStationId].nMask       := 0;
    _stState[_nStationId].nMoverId    := 0;

    IF (_stCtrl[_nStationId].eCmd = E_STATION_CTRL.STATION_MOVER_GONE)
    THEN
      _stState[_nStationId].eState    := E_STATION_STATE.STATION_DISABLE;

      IF (_eMessageLevel = E_MessageType.eMessageVerbose)
      THEN
        _stMsg.eType                  := _eMessageLevel;
        LogState(_stMsg.eType);
      END_IF
    END_IF
END_CASE
//-----------------------------------------------------------------------------
//-----------------------------------------------------------------------------
_sState                               := TO_STRING(_stState[_nStationId].eState);
//-----------------------------------------------------------------------------
//-----------------------------------------------------------------------------
// Error handling
//-----------------------------------------------------------------------------
CASE _stState[_nStationId].eState
OF
  //---------------------------------------------------------------------------
  //---------------------------------------------------------------------------
  E_STATION_STATE.STATION_ERROR_LIST_STATION_ID_WRONG:
    IF (_stCtrl[_nStationId].eCmd = E_STATION_CTRL.STATION_MOVER_OUT)
    THEN
      _nMoverDetected                 := _stMoverData.nMoverId;

      IF (_nMoverDetected < 1) OR
         (_nMoverDetected > MAX_MOVER)
      THEN
        // this MUST NOT happen
        _stState[_nStationId].eState  := E_STATION_STATE.STATION_ERROR_LIST_MOVER_ID_INVALID; // fatal error
        _stMsg.eType                  := E_MessageType.eMessageError;
        LogState(_stMsg.eType);

      ELSE
        // not for station; send mover out
        _stState[_nStationId].eState  := E_STATION_STATE.STATION_MOVER_OUT;

        IF (_eMessageLevel > E_MessageType.eMessageError)
        THEN
          _stMsg.eType                := E_MessageType.eMessageInfo;
          LogState(_stMsg.eType);
        END_IF
      END_IF

    ELSIF (_stCtrl[_nStationId].eCmd = E_STATION_CTRL.STATION_MOVER_ENTER)
    THEN
      // override wrong TargetStationId in List; start infeed of mover

      _nMoverDetected                 := _stMoverData.nMoverId;

      IF (_nMoverDetected < 1) OR
         (_nMoverDetected > MAX_MOVER)
      THEN
        // this MUST NOT happen
        _stState[_nStationId].eState  := E_STATION_STATE.STATION_ERROR_LIST_MOVER_ID_INVALID; // fatal error

        _stMsg.eType                  := E_MessageType.eMessageError;
        LogState(_stMsg.eType);

      ELSE
        _eStateProgress               := E_PROGRESS.PROGRESS_INIT;
        _stState[_nStationId].nMoverId:= TO_USINT(_nMoverDetected);
        _stState[_nStationId].nMask   := _stMoverData.nMask;
        _stState[_nStationId].eState  := E_STATION_STATE.STATION_MOVER_ENTER;

        IF (_eMessageLevel > E_MessageType.eMessageError)
        THEN
          _stMsg.eType                := E_MessageType.eMessageInfo;
          LogState(_stMsg.eType);
        END_IF
      END_IF
    END_IF

  //---------------------------------------------------------------------------
  //---------------------------------------------------------------------------
  E_STATION_STATE.STATION_ERROR_OUTFEED_TARGET_INVALID:
    // wait here until valid target is detected
    IF NOT (_stCtrl[_nStationId].nTargetStation < 1) AND  
       NOT (_stCtrl[_nStationId].nTargetStation > MAX_STATION)
    THEN
      _stState[_nStationId].eState    := E_STATION_STATE.STATION_MOVER_OUT;

      IF (_eMessageLevel > E_MessageType.eMessageError)
      THEN
        _stMsg.eType                  := E_MessageType.eMessageInfo;
        LogState(_stMsg.eType);
      END_IF
    END_IF

  //---------------------------------------------------------------------------
  //---------------------------------------------------------------------------
  E_STATION_STATE.STATION_ERROR_INFEED_ERROR:   // must be fixed by extern by using cyclic mover control
    IF (_stCtrl[_nStationId].eCmd = E_STATION_CTRL.STATION_MOVER_ENTER_RETRY)
    THEN
      _stState[_nStationId].eState    := E_STATION_STATE.STATION_DETECT_MOVER;   // return to start and wait

      IF (_eMessageLevel > E_MessageType.eMessageError)
      THEN
        _stMsg.eType                  := E_MessageType.eMessageInfo;
        LogState(_stMsg.eType);
      END_IF
    END_IF


  //---------------------------------------------------------------------------
  //---------------------------------------------------------------------------
  E_STATION_STATE.STATION_ERROR_OUTFEED_ERROR:  // must be fixed by extern by using cyclic mover control
    IF (_stCtrl[_nStationId].eCmd = E_STATION_CTRL.STATION_MOVER_OUT_RETRY)
    THEN
      MoverOut();
      _stState[_nStationId].eState  := E_STATION_STATE.STATION_MOVER_RELEASE;

      IF (_eMessageLevel > E_MessageType.eMessageError)
      THEN
        _stMsg.eType                  := E_MessageType.eMessageInfo;
        LogState(_stMsg.eType);
      END_IF

    ELSIF (_stCtrl[_nStationId].eCmd = E_STATION_CTRL.STATION_MOVER_GONE)
    THEN
      MoverOut();

      _stState[_nStationId].eState  := E_STATION_STATE.STATION_MOVER_WRITE_TARGET;

      IF (_eMessageLevel > E_MessageType.eMessageError)
      THEN
        _stMsg.eType                := E_MessageType.eMessageInfo;
        LogState(_stMsg.eType);
      END_IF
    END_IF

  //---------------------------------------------------------------------------
  // fatal errors
  //---------------------------------------------------------------------------
  E_STATION_STATE.STATION_ERROR_LIST_GET_HEAD_FAULT,
  E_STATION_STATE.STATION_ERROR_LIST_REMOVE_HEAD_FAULT,
  E_STATION_STATE.STATION_ERROR_LIST_ADD_TAIL_FAULT,
  E_STATION_STATE.STATION_ERROR_LIST_MOVER_ID_INVALID:
    _stMsg.eType                      := E_MessageType.eMessageError;
    LogState(_stMsg.eType);
    // yes, but why?
    // cannot be fixed by ctrl
    _eFatalError                      := _stState[_nStationId].eState;
    _stState[_nStationId].eState      := E_STATION_STATE.STATION_ERROR_FATAL;
    LogState(_stMsg.eType);

  //---------------------------------------------------------------------------
  //---------------------------------------------------------------------------
  E_STATION_STATE.STATION_ERROR_FATAL:
    // write to string for debugging
    _sState                           := concat(TO_STRING(_stState[_nStationId].eState), ': ');
    _sState                           := concat(_sState, TO_STRING(_eFatalError));
END_CASE
//-----------------------------------------------------------------------------
//-----------------------------------------------------------------------------
IF (_stState[_nStationId].nMoverId > 0) AND
   (_stState[_nStationId].nMoverId < MAX_MOVER+1)
THEN
  _stState[_nStationId].rMoverModPos  := _Mover[_stState[_nStationId].nMoverId].NcToPlc.ModuloActPos;
ELSE
  _stState[_nStationId].rMoverModPos  := 0.0;
END_IF
//-----------------------------------------------------------------------------
//-----------------------------------------------------------------------------
_stState[_nStationId].nQueue          := TO_USINT(_ItfStation[_nStationId].Count);
//-----------------------------------------------------------------------------
//-----------------------------------------------------------------------------
END_METHOD

METHOD PRIVATE DelBitWord : WORD
VAR_INPUT
  inVal   : WORD;
  bitNo   : DINT;
END_VAR
VAR
  wConst : WORD := 1;
END_VAR
IF ( inVal AND SHL( wConst, TO_SINT(bitNo) MOD 16 ) ) > 0 THEN
  DelBitWord := inVal XOR (SHL( wConst,TO_SINT(bitNo) MOD 16 ));
ELSE
  DelBitWord := inVal;
END_IF
END_METHOD

METHOD PRIVATE GetBitWord : BOOL
VAR_INPUT
  inVal   : WORD;
  bitNo   : DINT;
END_VAR
VAR
  wConst : WORD := 1;
END_VAR
IF ( inVal AND SHL( wConst,TO_SINT(bitNo) MOD 16 ) ) > 0
THEN
  GetBitWord := TRUE;
ELSE
  GetBitWord := FALSE;
END_IF
END_METHOD

METHOD Init : e_progress
VAR_INPUT
END_VAR
// check pointer and interface
IF NOT Check() THEN Init := e_progress.PROGRESS_ERROR; RETURN; END_IF

_stState[_nStationId].nMask       := 0;
_stState[_nStationId].nMoverId    := 0;

_eFatalError                      := E_STATION_STATE.STATION_ERROR_NULL;

_stState[_nStationId].eState      := E_STATION_STATE.STATION_INIT;
_sState                           := TO_STRING(_stState[_nStationId].eState);

IF _ItfStation[_nStationId].InitList()
THEN
  IF (_eMessageLevel = E_MessageType.eMessageVerbose)
  THEN
    _stMsg.eType                  := E_MessageType.eMessageVerbose;
    _stMsg.eSubdevice             := Stationstate;
    _stMsg.iErrorNumber           := 0;
    _stMsg.sText                  := concat('_ItfStation.InitList', ': ');
    _stMsg.sText                  := concat(_stMsg.sText, TO_STRING(E_PROGRESS.PROGRESS_DONE));
    //f_MessageSet(_stMsg);
  END_IF

  Init                            := E_PROGRESS.PROGRESS_DONE;

ELSE
    _stMsg.eType                  := E_MessageType.eMessageError;
    _stMsg.eSubdevice             := Stationstate;
    _stMsg.iErrorNumber           := 0;
    _stMsg.sText                  := concat('_ItfStation.InitList', ': ');
    _stMsg.sText                  := concat(_stMsg.sText, TO_STRING(E_PROGRESS.PROGRESS_ERROR));
    f_MessageSet(_stMsg);

  Init                            := e_progress.PROGRESS_ERROR;
END_IF
END_METHOD

PROPERTY ItfMover : reference to ARRAY[1..MAX_MOVER] OF I_XtsTransport_Mover
SET
_ItfMover ref= ItfMover;
END_SET
END_PROPERTY

PROPERTY ItfStations : reference to ARRAY[1..MAX_STATION] OF I_Station_LinkedList
SET
_ItfStation ref= ItfStations;
END_SET
END_PROPERTY

METHOD LogState
VAR_INPUT
  eType       : E_MessageType;
END_VAR
_stMsg.eType                := eType;
_stMsg.eSubdevice           := Stationstate;
_stMsg.iErrorNumber         := _stState[_nStationId].nMoverId;
_stMsg.sText                := TO_STRING(_stState[_nStationId].eState);
f_MessageSet(_stMsg);
END_METHOD

PROPERTY MessageLevel : e_messagetype
SET
_eMessageLevel := MessageLevel;
END_SET
END_PROPERTY

METHOD PRIVATE MoveData // prepares movement to PostStop[_nNest] in station
// build WorkPos from parameter, static station data and information on mover
_stInfeed.rPos            := _stParameter[_nStationId].rPosWait
                          +  _stParameter[_nStationId].rPosStop[_nNest]
                          +  _stMoverData.rOffset
                          +  _rMoverOffset[_nStationId][_stMoverData.nMoverId][_nNest];

_stInfeed.rVelo           := _stParameter[_nStationId].rVelo;
_stInfeed.rAcc            := _stParameter[_nStationId].rAccDec;
_stInfeed.rJerk           := _stParameter[_nStationId].rJerk;
_stInfeed.rGap            := _stParameter[_nStationId].rGap;
_stInfeed.rDistance       := _stParameter[_nStationId].rReleaseDistance;
_stInfeed.rDelta          := TargetWindow;

// init method
_ItfMover[_stState[_nStationId].nMoverId].MoveToPosCa(FALSE, _stInfeed);

// clear substate
_eStateProgress           := E_PROGRESS.PROGRESS_INIT;
END_METHOD

PROPERTY Mover : reference TO ARRAY[1..MAX_MOVER] OF AXIS_REF;
SET
_Mover ref= Mover;
END_SET
END_PROPERTY

PROPERTY MoverOffset : reference TO ARRAY[1..MAX_STATION]  OF T_NEST_OFFSET
SET
_rMoverOffset ref= MoverOffset;
END_SET
END_PROPERTY

METHOD PRIVATE MoverOut // prepares mover data for sending to target station
// build data for sending mover to target station

// who am I sending?
_stMoverDataSend.nMoverId         := _stState[_nStationId].nMoverId;

// get optional information about nests to work
_stMoverDataSend.nMask            := _stCtrl[_nStationId].nMask;

// get optional offset
_stMoverDataSend.rOffset          := _stCtrl[_nStationId].rOffset;

// get target station
_stMoverDataSend.nTargetStation   := _stCtrl[_nStationId].nTargetStation;

// get position of target
_stOutfeed.rPos                   := _stParameter[_stMoverDataSend.nTargetStation].rPosWait;

IF (_stOutfeed.rPos - _Mover[_stMoverDataSend.nMoverId].NcToPlc.ModuloActPos < 0)
THEN
  // only forward, never back
  _stOutfeed.rPos             := _stOutfeed.rPos 
                              +  _ItfMover[_stMoverDataSend.nMoverId].RailLength;
END_IF

_stOutfeed.rVelo              := _stParameter[_nStationId].rVelo;
_stOutfeed.rAcc               := _stParameter[_nStationId].rAccDec;
_stOutfeed.rJerk              := _stParameter[_nStationId].rJerk;
_stOutfeed.rGap               := _stParameter[_nStationId].rGap;
_stOutfeed.rDistance          := _stParameter[_nStationId].rReleaseDistance;

// init method for sending
_ItfMover[_stMoverDataSend.nMoverId].SendToModuloPosCa(FALSE, _stOutfeed);
END_METHOD

METHOD PRIVATE SetBitWord : WORD
VAR_INPUT
  inVal   : WORD;
  bitNo   : DINT;
END_VAR
VAR
  wConst  : WORD := 1;
END_VAR
SetBitWord := inVal OR SHL( wConst,TO_SINT(bitNo) MOD 16 );
END_METHOD

PROPERTY State : reference to ARRAY[1..MAX_STATION] OF ST_STATION_STATE
SET
_stState ref= State;
END_SET
END_PROPERTY

PROPERTY StationId : uint
GET
StationId := _nStationId;
END_GET
SET
_nStationId := StationId;
END_SET
END_PROPERTY

PROPERTY StationParameter : reference TO ARRAY[1..MAX_STATION]  OF ST_STATION_PARAMETER
SET
_stParameter ref= StationParameter;
END_SET
END_PROPERTY

PROPERTY TargetWindow : lreal
GET
TargetWindow := SEL((_stInfeed.rDelta < 0.05), _stInfeed.rDelta, 0.1);
END_GET
SET
_stInfeed.rDelta := SEL((TargetWindow < 0.05), TargetWindow, 0.1);
END_SET
END_PROPERTY

END_FUNCTION_BLOCK

// ---- XTS/CaGroup/FB_CaGroup.TcPOU
//---------------------------------------------------------------------------------------------------------------
//
//  HAUD 2023.12.13
//
//
//  fb_CaGroup
//  - handles CA group states
//  - add mover to group
//  - remove mover from group
//  - clear group error
//  - startup procedure for getting group ready to work
//
//
//  VAR INPUT / OUTPUT --> see properties
//
//---------------------------------------------------------------------------------------------------------------//
// This SOFTWARE is provided as an Exemple by THE PROVIDER "as is" and "with all faults." THE PROVIDER makes no  //
// representations or warranties of any kind concerning the safety, suitability, lack of viruses, inaccuracies,  //
// typographical errors, or other harmful components of this SOFTWARE. There are inherent dangers in the use of  //
// any software, and you are solely responsible for determining whether this SOFTWARE is compatible with your    //
// equipment and other software installed on your equipment. You are also solely responsible for the protection  //
// of your equipment and backup of your data, and THE PROVIDER will not be liable for any damages you may suffer //
// in connection with using, modifying, or distributing this SOFTWARE.                                           //
//---------------------------------------------------------------------------------------------------------------//
FUNCTION_BLOCK FB_CaGroup	IMPLEMENTS I_XtsTransport_CaGroup
VAR CONSTANT
{attribute 'hide'} 
  GROUP_HALT_JERK             : LREAL := 500_000.0;
{attribute 'hide'} 
  GROUP_HALT_DEC              : LREAL :=  12_500.0;
END_VAR
VAR
  _eCheck                     : E_GROUP_CHECK;
  _bError                     : BOOL;

  _GroupRef                   : REFERENCE TO Tc3_McCoordinatedMotion.AXES_GROUP_REF;

  _AxisRefMover               : REFERENCE TO ARRAY[1..MAX_MOVER] OF Tc2_MC2.AXIS_REF;
  _MoverItf                   : REFERENCE TO ARRAY[1..MAX_MOVER] OF I_XtsTransport_Mover;  // mover methods

  _stMoveData                 : ST_MOVE_DATA; // dyn constraints for _MoverItf[i].Halt(Execute, stMoveData)

  // CA group fb instances
  _fbAddAxisGroup             : ARRAY[1..MAX_MOVER] OF Tc3_McCoordinatedMotion.MC_AddAxisToGroup;
  _fbRemoveAxisGroup          : ARRAY[1..MAX_MOVER] OF Tc3_McCoordinatedMotion.MC_RemoveAxisFromGroup;

  _fbGroupDisable             : Tc3_McCoordinatedMotion.MC_GroupDisable;
  _fbGroupEnable              : Tc3_McCoordinatedMotion.MC_GroupEnable;
  _fbGroupErrorRead           : Tc3_McCoordinatedMotion.MC_GroupReadError;
  _fbGroupStatusRead          : Tc3_McCoordinatedMotion.MC_GroupReadStatus;
  _fbGroupReset               : Tc3_McCoordinatedMotion.MC_GroupReset;
  _fbGroupStop                : Tc3_McCoordinatedMotion.MC_GroupStop;

  _stGroupInfo                : ST_GROUP_INFO;  // additional bits about the state of the CA group

  _rtrigGroupStatusRead,
  _rtrigGroupErrorRead        : Tc2_Standard.R_TRIG;

  _stMsg                      : ST_Message;
  _eMessageLevel              : E_MessageType;
END_VAR

METHOD AddAll : E_PROGRESS
VAR_INPUT
  Execute     : BOOL;
END_VAR
VAR_INST
  _nErrorId   : UDINT;
  _eState     : E_PROGRESS;

  _nMover     : UINT;
END_VAR
IF NOT Execute THEN _eState     := E_PROGRESS.PROGRESS_INIT; END_IF 
IF NOT Check() THEN AddAll := E_PROGRESS.PROGRESS_ERROR; RETURN; END_IF


CASE _eState
OF
  E_PROGRESS.PROGRESS_INIT:
    IF Execute
    THEN
      _nErrorId               := 0;
      _nMover                 := 1;

      IF (_stGroupInfo.AxisCount < MAX_MOVER)
      THEN
        _eState               := E_PROGRESS.PROGRESS_BUSY;

      ELSE
        _eState               := E_PROGRESS.PROGRESS_DONE;

        IF (_eMessageLevel = E_MessageType.eMessageVerbose)
        THEN
          _stMsg.eType        := E_MessageType.eMessageVerbose;
          _stMsg.eSubdevice   := e_Subdevice.fbGroupAddAxis;
          _stMsg.iErrorNumber := _nMover;
          _stMsg.sText        := TO_STRING(_eState);
          f_MessageSet(_stMsg);
        END_IF
      END_IF
    END_IF
END_CASE
//-----------------------------------------------------------------------------
//-----------------------------------------------------------------------------
CASE _eState
OF
  E_PROGRESS.PROGRESS_BUSY:
    IF (_eMessageLevel = E_MessageType.eMessageVerbose)
    THEN
      _stMsg.eType            := E_MessageType.eMessageVerbose;
      _stMsg.eSubdevice       := e_Subdevice.fbGroupAddAxis;
      _stMsg.iErrorNumber     := _nMover;
      _stMsg.sText            := TO_STRING(_eState);
      f_MessageSet(_stMsg);
    END_IF

    _eState                   := E_PROGRESS.PROGRESS_PREPARE;
    _fbAddAxisGroup[_nMover](
                AxesGroup     := _GroupRef, 
                Axis          := _AxisRefMover[_nMover], 
                Execute       := FALSE, 
                IdentInGroup  := UDINT_TO_IDENTINGROUP(_AxisRefMover[_nMover].NcToPlc.AxisId));
END_CASE
//-----------------------------------------------------------------------------
//-----------------------------------------------------------------------------
CASE _eState
OF
  E_PROGRESS.PROGRESS_PREPARE:
    _fbAddAxisGroup[_nMover](
                AxesGroup     := _GroupRef, 
                Axis          := _AxisRefMover[_nMover], 
                Execute       := TRUE, 
                IdentInGroup  := UDINT_TO_IDENTINGROUP(_AxisRefMover[_nMover].NcToPlc.AxisId));

    IF (_fbAddAxisGroup[_nMover].Error)
    THEN
      _eState                 := E_PROGRESS.PROGRESS_ERROR;
      _nErrorId               := _fbAddAxisGroup[_nMover].ErrorId;

      _stMsg.eType            := E_MessageType.eMessageError;
      _stMsg.eSubdevice       := e_Subdevice.fbGroupAddAxis;
      _stMsg.iErrorNumber     := _nErrorId;
      _stMsg.sText            := TO_STRING(_eState);
      f_MessageSet(_stMsg);

    ELSIF (_fbAddAxisGroup[_nMover].Done)
    THEN
      _eState                 := E_PROGRESS.PROGRESS_CHECK;

      IF (_eMessageLevel = E_MessageType.eMessageVerbose)
      THEN
        _stMsg.eType          := E_MessageType.eMessageVerbose;
        _stMsg.eSubdevice     := e_Subdevice.fbGroupAddAxis;
        _stMsg.iErrorNumber   := _nMover;
        _stMsg.sText          := TO_STRING(_eState);
        f_MessageSet(_stMsg);
      END_IF
    END_IF
END_CASE
//-----------------------------------------------------------------------------
//-----------------------------------------------------------------------------
CASE _eState
OF
  E_PROGRESS.PROGRESS_CHECK:
    _eState                   := E_PROGRESS.PROGRESS_OCCUPIED;
    _fbAddAxisGroup[_nMover](
                AxesGroup     := _GroupRef, 
                Axis          := _AxisRefMover[_nMover], 
                Execute       := FALSE, 
                IdentInGroup  := UDINT_TO_IDENTINGROUP(_AxisRefMover[_nMover].NcToPlc.AxisId));
END_CASE
//-----------------------------------------------------------------------------
//-----------------------------------------------------------------------------
CASE _eState
OF
  E_PROGRESS.PROGRESS_OCCUPIED:
    IF (_nMover > MAX_MOVER-1)
    THEN
      _eState                 := E_PROGRESS.PROGRESS_DONE;

      IF (_eMessageLevel > E_MessageType.eMessageError)
      THEN
        _stMsg.eType          := E_MessageType.eMessageInfo;
        _stMsg.eSubdevice     := e_Subdevice.fbGroupAddAxis;
        _stMsg.iErrorNumber   := MAX_MOVER;
        _stMsg.sText          := TO_STRING(_eState);
        f_MessageSet(_stMsg);
      END_IF
    ELSE
      _nMover                 := _nMover + 1;
      _eState                 := E_PROGRESS.PROGRESS_BUSY;
    END_IF
END_CASE
//-----------------------------------------------------------------------------
//-----------------------------------------------------------------------------

AddAll                   := _eState;
END_METHOD

PROPERTY AxisRef : REFERENCE TO ARRAY[1..MAX_MOVER] OF Tc2_MC2.AXIS_REF
SET
_AxisRefMover REF= AxisRef;
END_SET
END_PROPERTY

METHOD PROTECTED Check : BOOL

IF NOT __ISVALIDREF(_GroupRef)
THEN
  _eCheck                     := E_GROUP_CHECK.CHECK_GROUP_REF_INVALID;
  RETURN;
END_IF

IF NOT __ISVALIDREF(_AxisRefMover)
THEN
  _eCheck                     := E_GROUP_CHECK.CHECK_AXIS_REF_INVALID;
  RETURN;
END_IF

IF NOT __ISVALIDREF(_MoverItf)
THEN
  _eCheck                     := E_GROUP_CHECK.CHECK_Mover_ITF_REF_INVALID;
  RETURN;
END_IF

_eCheck                       := E_GROUP_CHECK.CHECK_DONE;
Check                         := TRUE;
END_METHOD

METHOD Disable : E_PROGRESS
VAR_INPUT
  Execute     : BOOL;
END_VAR
VAR_INST
  _nErrorId   : UDINT;
  _eState     : E_PROGRESS;

  _nMover     : UINT;
END_VAR
IF NOT Execute THEN _eState       := E_PROGRESS.PROGRESS_INIT; END_IF 
IF NOT Check() THEN Disable  := E_PROGRESS.PROGRESS_ERROR; RETURN; END_IF


CASE _eState
OF
  E_PROGRESS.PROGRESS_INIT:
    IF Execute
    THEN
      _nErrorId               := 0;
      _nMover                 := 1;
      _eState                 := E_PROGRESS.PROGRESS_BUSY;
    END_IF
END_CASE
//-----------------------------------------------------------------------------
//-----------------------------------------------------------------------------
CASE _eState
OF
  E_PROGRESS.PROGRESS_BUSY:
    IF (_stGroupInfo.CaGroupState = E_CA_GROUP_STATE.mcGroupStateDisabled)
    THEN
      _eState                 := E_PROGRESS.PROGRESS_DONE;

      IF (_eMessageLevel = E_MessageType.eMessageVerbose)
      THEN
        _stMsg.eType          := E_MessageType.eMessageVerbose;
        _stMsg.eSubdevice     := e_Subdevice.fbGroupDisable;
        _stMsg.iErrorNumber   := _nErrorId;
        _stMsg.sText          := TO_STRING(_eState);
        f_MessageSet(_stMsg);
      END_IF
    ELSE
      _eState                 := E_PROGRESS.PROGRESS_PREPARE;
      _fbGroupDisable(
                AxesGroup     := _GroupRef, 
                Execute       := FALSE);

      _fbGroupReset(
                AxesGroup     := _GroupRef, 
                Execute       := FALSE);
  
      IF (_eMessageLevel = E_MessageType.eMessageVerbose)
      THEN
        _stMsg.eType          := E_MessageType.eMessageVerbose;
        _stMsg.eSubdevice     := e_Subdevice.fbGroupDisable;
        _stMsg.iErrorNumber   := _nErrorId;
        _stMsg.sText          := TO_STRING(_eState);
        f_MessageSet(_stMsg);
      END_IF
    END_IF
END_CASE
//-----------------------------------------------------------------------------
//-----------------------------------------------------------------------------
CASE _eState
OF
  E_PROGRESS.PROGRESS_PREPARE:
    _fbGroupReset(
                AxesGroup     := _GroupRef, 
                Execute       := TRUE);

    IF (_fbGroupReset.Error)
    THEN
      _eState                 := E_PROGRESS.PROGRESS_ERROR;
      _nErrorId               := _fbGroupReset.ErrorId;

      _stMsg.eType            := E_MessageType.eMessageError;
      _stMsg.eSubdevice       := e_Subdevice.fbGroupReset;
      _stMsg.iErrorNumber     := _nErrorId;
      _stMsg.sText            := TO_STRING(_eState);
      f_MessageSet(_stMsg);

      _fbGroupReset(
                AxesGroup     := _GroupRef, 
                Execute       := FALSE);
    ELSE
      IF (_fbGroupReset.Done)
      THEN
        _eState               := E_PROGRESS.PROGRESS_STARTUP;
        _fbGroupReset(
                AxesGroup     := _GroupRef, 
                Execute       := FALSE);
      END_IF
    END_IF
END_CASE
//-----------------------------------------------------------------------------
//-----------------------------------------------------------------------------
CASE _eState
OF
  E_PROGRESS.PROGRESS_STARTUP:
    _fbGroupDisable(
              AxesGroup       := _GroupRef, 
              Execute         := TRUE); 

    IF (_fbGroupDisable.Error)
    THEN
      _eState                 := E_PROGRESS.PROGRESS_ERROR;
      _nErrorId               := _fbGroupDisable.ErrorId;

      _stMsg.eType            := E_MessageType.eMessageError;
      _stMsg.eSubdevice       := e_Subdevice.fbGroupDisable;
      _stMsg.iErrorNumber     := _nErrorId;
      _stMsg.sText            := TO_STRING(_eState);
      f_MessageSet(_stMsg);

      _fbGroupDisable(
              AxesGroup       := _GroupRef, 
              Execute         := FALSE); 


    ELSIF (_fbGroupDisable.Done)
    THEN
      _eState                 := E_PROGRESS.PROGRESS_DONE;

      IF (_eMessageLevel > E_MessageType.eMessageError)
      THEN
        _stMsg.eType          := E_MessageType.eMessageInfo;
        _stMsg.eSubdevice     := e_Subdevice.fbGroupDisable;
        _stMsg.iErrorNumber   := _nErrorId;
        _stMsg.sText          := TO_STRING(_eState);
        f_MessageSet(_stMsg);
      END_IF

      _fbGroupDisable(
              AxesGroup       := _GroupRef, 
              Execute         := FALSE); 
    END_IF
END_CASE
//-----------------------------------------------------------------------------
//-----------------------------------------------------------------------------

Disable                  := _eState;
END_METHOD

METHOD Enable : E_PROGRESS
VAR_INPUT
  Execute     : BOOL;
END_VAR
VAR_INST
  _nErrorId   : UDINT;
  _eState     : E_PROGRESS;

  _nMover     : UINT;
END_VAR
IF NOT Execute THEN _eState       := E_PROGRESS.PROGRESS_INIT; END_IF 
IF NOT Check() THEN Enable   := E_PROGRESS.PROGRESS_ERROR; RETURN; END_IF


CASE _eState
OF
  E_PROGRESS.PROGRESS_INIT:
    IF Execute
    THEN
      _nErrorId               := 0;
      _nMover                 := 1;
      _eState                 := E_PROGRESS.PROGRESS_BUSY;
    END_IF
END_CASE
//-----------------------------------------------------------------------------
//-----------------------------------------------------------------------------
CASE _eState
OF
  E_PROGRESS.PROGRESS_BUSY:
    _eState                   := E_PROGRESS.PROGRESS_PREPARE;
    _fbGroupEnable(
                AxesGroup     := _GroupRef, 
                Execute       := FALSE);

    IF (_eMessageLevel = E_MessageType.eMessageVerbose)
    THEN
      _stMsg.eType            := E_MessageType.eMessageVerbose;
      _stMsg.eSubdevice       := e_Subdevice.fbGroupEnable;
      _stMsg.iErrorNumber     := _nErrorId;
      _stMsg.sText            := TO_STRING(_eState);
      f_MessageSet(_stMsg);
    END_IF
END_CASE
//-----------------------------------------------------------------------------
//-----------------------------------------------------------------------------
CASE _eState
OF
  E_PROGRESS.PROGRESS_PREPARE:
    _fbGroupEnable(
                AxesGroup     := _GroupRef, 
                Execute       := TRUE);

    IF (_fbGroupEnable.Error)
    THEN
      _eState                 := E_PROGRESS.PROGRESS_ERROR;
      _nErrorId               := _fbGroupEnable.ErrorId;

      _stMsg.eType            := E_MessageType.eMessageError;
      _stMsg.eSubdevice       := e_Subdevice.fbGroupEnable;
      _stMsg.iErrorNumber     := _nErrorId;
      _stMsg.sText            := TO_STRING(_eState);
      f_MessageSet(_stMsg);

      _fbGroupEnable(
                AxesGroup     := _GroupRef, 
                Execute       := FALSE);

    ELSIF (_fbGroupEnable.Done)
    THEN
      _eState                 := E_PROGRESS.PROGRESS_DONE;

      IF (_eMessageLevel > E_MessageType.eMessageError)
      THEN
        _stMsg.eType          := E_MessageType.eMessageInfo;
        _stMsg.eSubdevice     := e_Subdevice.fbGroupEnable;
        _stMsg.iErrorNumber   := _nErrorId;
        _stMsg.sText          := TO_STRING(_eState);
        f_MessageSet(_stMsg);
      END_IF
      _fbGroupEnable(
                AxesGroup     := _GroupRef, 
                Execute       := FALSE);
    END_IF
END_CASE
//-----------------------------------------------------------------------------
//-----------------------------------------------------------------------------

Enable                   := _eState;
END_METHOD

PROPERTY GroupInfo : reference to ST_GROUP_INFO
GET
GroupInfo REF= _stGroupInfo;
END_GET
END_PROPERTY

PROPERTY GroupRef : reference to Tc3_McCoordinatedMotion.AXES_GROUP_REF
GET
GroupRef REF= _GroupRef;
END_GET
SET
_GroupRef REF= GroupRef;
END_SET
END_PROPERTY

METHOD InfoCycle : DWORD
VAR_INPUT
  EnableCycle          : BOOL;
END_VAR
VAR_INST
  _nErrorIdADS,
  _nErrorIdRead   : UDINT;

  _nIdx           : udint;
END_VAR
IF NOT Check() THEN RETURN; END_IF

_stMsg.eDevice                              := e_Device.CaGroup;

//-----------------------------------------------------------------------------------------------
// cyclic CA group
//-----------------------------------------------------------------------------------------------
_fbGroupStatusRead(
              AxesGroup                     := _GroupRef, 
              Enable                        := EnableCycle, 
              Valid                         => _stGroupInfo.GroupStatusValid, 
              Busy                          => _stGroupInfo.GroupStatusBusy, 
              GroupMoving                   => _stGroupInfo.GroupMoving, 
              GroupHoming                   => _stGroupInfo.GroupHoming, 
              GroupErrorStop                => _stGroupInfo.GroupErrorStop, 
              GroupNotReady                 => _stGroupInfo.GroupNotReady, 
              GroupStandby                  => _stGroupInfo.GroupStandby, 
              GroupStopping                 => _stGroupInfo.GroupStopping, 
              GroupDisabled                 => _stGroupInfo.GroupDisabled, 
              AllAxesStanding               => _stGroupInfo.AllAxesStanding, 
              ConstantVelocity              => _stGroupInfo.ConstantVelocity, 
              Accelerating                  => _stGroupInfo.Accelerating, 
              Decelerating                  => _stGroupInfo.Decelerating, 
              InPosition                    => _stGroupInfo.InPosition, 
              Error                         => _stGroupInfo.GroupError, 
              ErrorId                       => );

_fbGroupErrorRead(
              AxesGroup                     := _GroupRef, 
              Enable                        := EnableCycle, 
              ErrorId                       => , 
              GroupErrorId                  => _stGroupInfo.GroupErrorId);


_stGroupInfo.AxisCount                      := _GroupRef.NcToPlc.CA.Common.GroupAxesCount;
_stGroupInfo.CaGroupOID                     := _GroupRef.NcToPlc.CA.Common.GroupOID;
_stGroupInfo.CaGroupState                   := TO_UINT(_GroupRef.NcToPlc.CA.Common.GroupStatus.State);

_stGroupInfo.AxisCountEnabled               := 0;
FOR _nIdx := 1 TO MAX_MOVER
DO
  IF (_AxisRefMover[_nIdx].Status.ControlLoopClosed)
  THEN
    _stGroupInfo.AxisCountEnabled           := _stGroupInfo.AxisCountEnabled + 1;
  END_IF
END_FOR	
			  
// fetch internal fb error
_rtrigGroupErrorRead(CLK                    := _fbGroupErrorRead.Error);
IF _rtrigGroupErrorRead.Q
THEN
  _nErrorIdADS                              := _fbGroupErrorRead.ErrorId;

  _stMsg.eType                              := E_MessageType.eMessageError;
  _stMsg.eSubdevice                         := e_Subdevice.fbGroupErrorRead;
  _stMsg.iErrorNumber                       := _nErrorIdADS;
  _stMsg.sText                              := '';
  f_MessageSet(_stMsg);
END_IF

// Dyn constrainst for McHaltAll(method)
_stMoveData.rJerk                           := GROUP_HALT_JERK;
_stMoveData.rAcc                            := GROUP_HALT_DEC;
END_METHOD

METHOD McHaltAll : E_PROGRESS
VAR_INPUT
  Execute       : BOOL;
END_VAR
VAR_INST
  _nErrorId     : UDINT;
  _eState       : E_PROGRESS;
  _eResult      : E_PROGRESS;

  _nMover       : UINT;

  _nRepeat      : UINT;
END_VAR
IF NOT Execute 
THEN 
	_eState     := E_PROGRESS.PROGRESS_INIT; 
END_IF 
IF NOT Check() 
THEN 
	McHaltAll   := E_PROGRESS.PROGRESS_ERROR; 
	RETURN; 
END_IF


CASE _eState
OF
  E_PROGRESS.PROGRESS_INIT:
    IF Execute
    THEN
      _fbGroupStop(
              AxesGroup       := _GroupRef, 
              Execute         := FALSE, 
              Deceleration    := GROUP_HALT_DEC, 
              Jerk            := GROUP_HALT_JERK);

      _nErrorId               := 0;
      _nMover                 := 1;
      _eState                 := E_PROGRESS.PROGRESS_BUSY;
    END_IF
END_CASE

//-----------------------------------------------------------------------------
//-----------------------------------------------------------------------------
CASE _eState
OF
  E_PROGRESS.PROGRESS_BUSY:
    IF NOT (_stGroupInfo.CaGroupState = E_CA_GROUP_STATE.mcGroupStateMoving)
    THEN
      _eState                   := E_PROGRESS.PROGRESS_PREPARE;
    ELSE
      _fbGroupStop(
                AxesGroup       := _GroupRef, 
                Execute         := TRUE, 
                Deceleration    := GROUP_HALT_DEC, 
                Jerk            := GROUP_HALT_JERK);
  
      IF (_fbGroupStop.Error)
      THEN
        _stMsg.eType            := E_MessageType.eMessageError;
        _stMsg.eSubdevice       := e_Subdevice.fbGroupStop;
        _stMsg.iErrorNumber     := _fbGroupStop.ErrorId;
        _stMsg.sText            := TO_STRING(_eState);
        f_MessageSet(_stMsg);
  
        _nRepeat                := _nRepeat + 1;
        _eState                 := E_PROGRESS.PROGRESS_PREPARE;
      ELSE
        IF (_fbGroupStop.Done)
        THEN
          IF (_eMessageLevel = E_MessageType.eMessageVerbose)
          THEN
            _stMsg.eType        := E_MessageType.eMessageVerbose;
            _stMsg.eSubdevice   := e_Subdevice.fbGroupStop;
            _stMsg.iErrorNumber := MAX_MOVER;
            _stMsg.sText        := TO_STRING(_eState);
            f_MessageSet(_stMsg);
          END_IF
          _nRepeat              := 0;
          _eState               := E_PROGRESS.PROGRESS_PREPARE;
        END_IF
      END_IF
    END_IF
END_CASE

//-----------------------------------------------------------------------------
//-----------------------------------------------------------------------------
CASE _eState
OF
  E_PROGRESS.PROGRESS_PREPARE:
    _eState                   := E_PROGRESS.PROGRESS_WORKING;
    _fbGroupStop(
              AxesGroup       := _GroupRef, 
              Execute         := FALSE, 
              Deceleration    := GROUP_HALT_DEC, 
              Jerk            := GROUP_HALT_JERK);

    _eResult                  := _MoverItf[_nMover].Reset(FALSE);
    _eResult                  := _MoverItf[_nMover].Halt(FALSE, _stMoveData);
END_CASE
//-----------------------------------------------------------------------------
//-----------------------------------------------------------------------------
CASE _eState
OF
  E_PROGRESS.PROGRESS_WORKING:
    _eResult                  := _MoverItf[_nMover].Halt(TRUE, _stMoveData);

    IF (_eResult = E_PROGRESS.PROGRESS_DONE)
    THEN
      _eResult                := _MoverItf[_nMover].Halt(FALSE, _stMoveData);
      _eState                 := E_PROGRESS.PROGRESS_STARTUP;

    ELSIF (_eResult = E_PROGRESS.PROGRESS_ERROR)
    THEN
      _nErrorId               := _AxisRefMover[_nMover].NcToPlc.ErrorCode;
      _MoverItf[_nMover].Reset(TRUE);

      _stMsg.eType            := E_MessageType.eMessageError;
      _stMsg.eSubdevice       := e_Subdevice.fbHalt;
      _stMsg.iErrorNumber     := _nErrorId;
      _stMsg.sText            := concat( 'McHaltAll: ', TO_STRING(_eResult));
      _stMsg.sText            := concat(_stMsg.sText, ' MoverId: ');
      _stMsg.sText            := concat(_stMsg.sText, TO_STRING(_nMover));
      f_MessageSet(_stMsg);

      _eState                 := E_PROGRESS.PROGRESS_PREPARE;
    END_IF
END_CASE

//-----------------------------------------------------------------------------
//-----------------------------------------------------------------------------
CASE _eState
OF
  E_PROGRESS.PROGRESS_STARTUP:
    IF (_nMover > MAX_MOVER-1)
    THEN
      _eState                 := E_PROGRESS.PROGRESS_CHECK;
    ELSE
      _nMover                 := _nMover + 1;
      _eState                 := E_PROGRESS.PROGRESS_PREPARE;
    END_IF
END_CASE

//-----------------------------------------------------------------------------
//-----------------------------------------------------------------------------
CASE _eState
OF
  E_PROGRESS.PROGRESS_CHECK:
    _eState                   := E_PROGRESS.PROGRESS_DONE;

    IF (_eMessageLevel > E_MessageType.eMessageError)
    THEN
      _stMsg.eType            := E_MessageType.eMessageInfo;
      _stMsg.eSubdevice       := e_Subdevice.fbCaGroup;
      _stMsg.iErrorNumber     := MAX_MOVER;
      _stMsg.sText            := concat('McHaltAll: ', TO_STRING(_eState));
      f_MessageSet(_stMsg);
    END_IF
END_CASE
//-----------------------------------------------------------------------------
//-----------------------------------------------------------------------------
McHaltAll                     := _eState;
END_METHOD

